    |   movel([-0.082267, -1.492529, -2.487581, -0.732279, 1.570796, 1.488530],accel_mss,speed_ms,0,blend_radius_m)
    |   movel([-0.082969, -1.494588, -2.485777, -0.732025, 1.570796, 1.487827],accel_mss,speed_ms,0,blend_radius_m)
    |   movel([-0.083539, -1.496624, -2.483986, -0.731779, 1.570796, 1.487258],accel_mss,speed_ms,0,blend_radius_m)
    |   movel([-0.083978, -1.498631, -2.482215, -0.731544, 1.570796, 1.486818],accel_mss,speed_ms,0,blend_radius_m)
    |   movel([-0.084285, -1.500606, -2.480465, -0.731318, 1.570796, 1.486511],accel_mss,speed_ms,0,blend_radius_m)
    |   movel([-0.084466, -1.502546, -2.478740, -0.731103, 1.570796, 1.486331],accel_mss,speed_ms,0,blend_radius_m)
    |   movel([-0.084516, -1.504447, -2.477045, -0.730898, 1.570796, 1.486280],accel_mss,speed_ms,0,blend_radius_m)
    |   movel([-0.084436, -1.506303, -2.475383, -0.730703, 1.570796, 1.486361],accel_mss,speed_ms,0,blend_radius_m)
    |   movel([-0.084230, -1.508115, -2.473757, -0.730518, 1.570796, 1.486566],accel_mss,speed_ms,0,blend_radius_m)
    |   movel([-0.083899, -1.509875, -2.472171, -0.730343, 1.570796, 1.486898],accel_mss,speed_ms,0,blend_radius_m)
    |   movel([-0.083438, -1.511581, -2.470630, -0.730178, 1.570796, 1.487358],accel_mss,speed_ms,0,blend_radius_m)
    |   movel([-0.082854, -1.513231, -2.469135, -0.730023, 1.570796, 1.487942],accel_mss,speed_ms,0,blend_radius_m)
    |   movel([-0.082145, -1.514819, -2.467691, -0.729879, 1.570796, 1.488651],accel_mss,speed_ms,0,blend_radius_m)
    |   movel([-0.081311, -1.516345, -2.466301, -0.729743, 1.570796, 1.489485],accel_mss,speed_ms,0,blend_radius_m)
    |   movel([-0.079795, -1.518566, -2.464270, -0.729553, 1.570796, 1.491001],accel_mss,speed_ms,0,blend_radius_m)
    |   movel([-0.078055, -1.520599, -2.462405, -0.729385, 1.570796, 1.492742],accel_mss,speed_ms,0,blend_radius_m)
    |   movel([-0.076117, -1.522459, -2.460692, -0.729238, 1.570796, 1.494679],accel_mss,speed_ms,0,blend_radius_m)
    |   movel([-0.074001, -1.524162, -2.459119, -0.729108, 1.570796, 1.496795],accel_mss,speed_ms,0,blend_radius_m)
    |   movel([-0.071735, -1.525724, -2.457672, -0.728993, 1.570796, 1.499062],accel_mss,speed_ms,0,blend_radius_m)
    |   movel([-0.069341, -1.527159, -2.456340, -0.728890, 1.570796, 1.501456],accel_mss,speed_ms,0,blend_radius_m)
    |   movel([-0.066843, -1.528483, -2.455108, -0.728799, 1.570796, 1.503953],accel_mss,speed_ms,0,blend_radius_m)
    |   movel([-0.064261, -1.529706, -2.453967, -0.728716, 1.570796, 1.506535],accel_mss,speed_ms,0,blend_radius_m)
    |   movel([-0.058915, -1.531954, -2.451863, -0.728572, 1.570796, 1.511882],accel_mss,speed_ms,0,blend_radius_m)
    |   movel([-0.053475, -1.534068, -2.449878, -0.728443, 1.570796, 1.517321],accel_mss,speed_ms,0,blend_radius_m)
    |   movel([-0.049350, -1.535795, -2.448251, -0.728343, 1.570796, 1.521446],accel_mss,speed_ms,0,blend_radius_m)
    |   movel([-0.047922, -1.536279, -2.447794, -0.728316, 1.570796, 1.522874],accel_mss,speed_ms,0,blend_radius_m)
    |   movel([-0.045334, -1.536940, -2.447169, -0.728280, 1.570796, 1.525463],accel_mss,speed_ms,0,blend_radius_m)
    |   movel([-0.044798, -1.537178, -2.446944, -0.728267, 1.570796, 1.525998],accel_mss,speed_ms,0,blend_radius_m)
    |   movel([-0.044322, -1.537503, -2.446637, -0.728250, 1.570796, 1.526475],accel_mss,speed_ms,0,blend_radius_m)
    |   movel([-0.043916, -1.537944, -2.446219, -0.728226, 1.570796, 1.526880],accel_mss,speed_ms,0,blend_radius_m)
    |   movel([-0.043592, -1.538530, -2.445663, -0.728195, 1.570796, 1.527205],accel_mss,speed_ms,0,blend_radius_m)
    |   movel([-0.043368, -1.539293, -2.444940, -0.728156, 1.570796, 1.527428],accel_mss,speed_ms,0,blend_radius_m)
    |   movel([-0.043314, -1.540103, -2.444171, -0.728116, 1.570796, 1.527483],accel_mss,speed_ms,0,blend_radius_m)
    |   movel([-0.043411, -1.540949, -2.443366, -0.728074, 1.570796, 1.527385],accel_mss,speed_ms,0,blend_radius_m)
    |   movel([-0.043649, -1.541827, -2.442530, -0.728033, 1.570796, 1.527148],accel_mss,speed_ms,0,blend_radius_m)
    |   movel([-0.044011, -1.542723, -2.441675, -0.727991, 1.570796, 1.526786],accel_mss,speed_ms,0,blend_radius_m)
    |   movel([-0.045056, -1.544546, -2.439931, -0.727912, 1.570796, 1.525740],accel_mss,speed_ms,0,blend_radius_m)
    |   movel([-0.045713, -1.545455, -2.439061, -0.727874, 1.570796, 1.525083],accel_mss,speed_ms,0,blend_radius_m)
    |   movel([-0.047218, -1.547224, -2.437361, -0.727804, 1.570796, 1.523578],accel_mss,speed_ms,0,blend_radius_m)
    |   movel([-0.048899, -1.548876, -2.435770, -0.727744, 1.570796, 1.521898],accel_mss,speed_ms,0,blend_radius_m)
    |   movel([-0.050641, -1.550343, -2.434352, -0.727694, 1.570796, 1.520155],accel_mss,speed_ms,0,blend_radius_m)
    |   movel([-0.052345, -1.551562, -2.433172, -0.727655, 1.570796, 1.518451],accel_mss,speed_ms,0,blend_radius_m)
    |   movel([-0.055003, -1.553125, -2.431656, -0.727608, 1.570796, 1.515794],accel_mss,speed_ms,0,blend_radius_m)
    |   movel([-0.056377, -1.553814, -2.430986, -0.727589, 1.570796, 1.514419],accel_mss,speed_ms,0,blend_radius_m)
    |   movel([-0.057771, -1.554438, -2.430379, -0.727572, 1.570796, 1.513025],accel_mss,speed_ms,0,blend_radius_m)
    |   movel([-0.060603, -1.555491, -2.429353, -0.727545, 1.570796, 1.510193],accel_mss,speed_ms,0,blend_radius_m)
    |   movel([-0.063453, -1.556276, -2.428587, -0.727526, 1.570796, 1.507344],accel_mss,speed_ms,0,blend_radius_m)
    |   movel([-0.066275, -1.556782, -2.428092, -0.727515, 1.570796, 1.504521],accel_mss,speed_ms,0,blend_radius_m)
    |   movel([-0.069020, -1.557000, -2.427879, -0.727510, 1.570796, 1.501776],accel_mss,speed_ms,0,blend_radius_m)
    |   movel([-0.070351, -1.556996, -2.427883, -0.727510, 1.570796, 1.500445],accel_mss,speed_ms,0,blend_radius_m)
    |   movel([-0.072900, -1.556759, -2.428115, -0.727515, 1.570796, 1.497896],accel_mss,speed_ms,0,blend_radius_m)
    |   movel([-0.074106, -1.556521, -2.428347, -0.727521, 1.570796, 1.496690],accel_mss,speed_ms,0,blend_radius_m)
    |   movel([-0.075629, -1.556091, -2.428768, -0.727531, 1.570796, 1.495168],accel_mss,speed_ms,0,blend_radius_m)
    |   movel([-0.077066, -1.555548, -2.429297, -0.727544, 1.570796, 1.493731],accel_mss,speed_ms,0,blend_radius_m)
    |   movel([-0.078425, -1.554908, -2.429921, -0.727560, 1.570796, 1.492372],accel_mss,speed_ms,0,blend_radius_m)
    |   movel([-0.079719, -1.554187, -2.430624, -0.727579, 1.570796, 1.491077],accel_mss,speed_ms,0,blend_radius_m)
    |   movel([-0.082152, -1.552560, -2.432204, -0.727624, 1.570796, 1.488644],accel_mss,speed_ms,0,blend_radius_m)
    |   movel([-0.084447, -1.550793, -2.433917, -0.727679, 1.570796, 1.486349],accel_mss,speed_ms,0,blend_radius_m)
    |   movel([-0.087214, -1.548474, -2.436157, -0.727758, 1.570796, 1.483583],accel_mss,speed_ms,0,blend_radius_m)
    |   movel([-0.089858, -1.546009, -2.438528, -0.727852, 1.570796, 1.480939],accel_mss,speed_ms,0,blend_radius_m)
    |   movel([-0.092354, -1.543396, -2.441032, -0.727961, 1.570796, 1.478443],accel_mss,speed_ms,0,blend_radius_m)
    |   movel([-0.094679, -1.540631, -2.443668, -0.728090, 1.570796, 1.476118],accel_mss,speed_ms,0,blend_radius_m)
    |   movel([-0.096807, -1.537710, -2.446441, -0.728238, 1.570796, 1.473989],accel_mss,speed_ms,0,blend_radius_m)
    |   movel([-0.098711, -1.534629, -2.449349, -0.728410, 1.570796, 1.472086],accel_mss,speed_ms,0,blend_radius_m)
    |   movel([-0.100365, -1.531386, -2.452395, -0.728608, 1.570796, 1.470431],accel_mss,speed_ms,0,blend_radius_m)
    |   movel([-0.101745, -1.527976, -2.455580, -0.728833, 1.570796, 1.469052],accel_mss,speed_ms,0,blend_radius_m)
    |   movel([-0.102598, -1.525304, -2.458061, -0.729023, 1.570796, 1.468199],accel_mss,speed_ms,0,blend_radius_m)
    |   movel([-0.103327, -1.522453, -2.460698, -0.729238, 1.570796, 1.467470],accel_mss,speed_ms,0,blend_radius_m)
    |   movel([-0.103895, -1.519449, -2.463461, -0.729479, 1.570796, 1.466901],accel_mss,speed_ms,0,blend_radius_m)
    |   movel([-0.104269, -1.516327, -2.466317, -0.729745, 1.570796, 1.466527],accel_mss,speed_ms,0,blend_radius_m)
    |   movel([-0.104412, -1.513119, -2.469236, -0.730034, 1.570796, 1.466384],accel_mss,speed_ms,0,blend_radius_m)
    |   movel([-0.104286, -1.509858, -2.472187, -0.730345, 1.570796, 1.466511],accel_mss,speed_ms,0,blend_radius_m)
    |   movel([-0.103856, -1.506574, -2.475141, -0.730675, 1.570796, 1.466940],accel_mss,speed_ms,0,blend_radius_m)
    |   movel([-0.103514, -1.504934, -2.476609, -0.730846, 1.570796, 1.467282],accel_mss,speed_ms,0,blend_radius_m)
    |   movel([-0.103083, -1.503302, -2.478066, -0.731020, 1.570796, 1.467714],accel_mss,speed_ms,0,blend_radius_m)
    |   movel([-0.102065, -1.500231, -2.480797, -0.731361, 1.570796, 1.468731],accel_mss,speed_ms,0,blend_radius_m)
    |   movel([-0.100816, -1.497139, -2.483531, -0.731718, 1.570796, 1.469980],accel_mss,speed_ms,0,blend_radius_m)
    |   movel([-0.099340, -1.494040, -2.486258, -0.732092, 1.570796, 1.471456],accel_mss,speed_ms,0,blend_radius_m)
    |   movel([-0.097645, -1.490946, -2.488963, -0.732480, 1.570796, 1.473151],accel_mss,speed_ms,0,blend_radius_m)
    |   movel([-0.095732, -1.487871, -2.491638, -0.732881, 1.570796, 1.475065],accel_mss,speed_ms,0,blend_radius_m)
    |   movel([-0.093611, -1.484830, -2.494267, -0.733292, 1.570796, 1.477185],accel_mss,speed_ms,0,blend_radius_m)
    |   movel([-0.091286, -1.481838, -2.496841, -0.733710, 1.570796, 1.479510],accel_mss,speed_ms,0,blend_radius_m)
    |   movel([-0.088762, -1.478910, -2.499346, -0.734134, 1.570796, 1.482034],accel_mss,speed_ms,0,blend_radius_m)
    |   movel([-0.092940, -1.473333, -2.504079, -0.734977, 1.570796, 1.477856],accel_mss,speed_ms,0,blend_radius_m)
    |   movel([-0.095041, -1.470536, -2.506435, -0.735418, 1.570796, 1.475755],accel_mss,speed_ms,0,blend_radius_m)
    |   movel([-0.097004, -1.467625, -2.508873, -0.735890, 1.570796, 1.473792],accel_mss,speed_ms,0,blend_radius_m)
    |   movel([-0.098264, -1.465308, -2.510805, -0.736276, 1.570796, 1.472533],accel_mss,speed_ms,0,blend_radius_m)
    |   movel([-0.099276, -1.462829, -2.512862, -0.736697, 1.570796, 1.471520],accel_mss,speed_ms,0,blend_radius_m)
    |   movel([-0.100052, -1.460205, -2.515030, -0.737154, 1.570796, 1.470745],accel_mss,speed_ms,0,blend_radius_m)
    |   movel([-0.100596, -1.457445, -2.517298, -0.737646, 1.570796, 1.470200],accel_mss,speed_ms,0,blend_radius_m)
    |   movel([-0.100917, -1.454564, -2.519654, -0.738172, 1.570796, 1.469879],accel_mss,speed_ms,0,blend_radius_m)
    |   movel([-0.101020, -1.451573, -2.522084, -0.738731, 1.570796, 1.469776],accel_mss,speed_ms,0,blend_radius_m)
    |   movel([-0.100913, -1.448486, -2.524579, -0.739323, 1.570796, 1.469883],accel_mss,speed_ms,0,blend_radius_m)
    |   movel([-0.100604, -1.445317, -2.527125, -0.739946, 1.570796, 1.470192],accel_mss,speed_ms,0,blend_radius_m)
    |   movel([-0.100098, -1.442082, -2.529709, -0.740598, 1.570796, 1.470699],accel_mss,speed_ms,0,blend_radius_m)
    |   movel([-0.099400, -1.438790, -2.532321, -0.741278, 1.570796, 1.471396],accel_mss,speed_ms,0,blend_radius_m)
    |   movel([-0.098520, -1.435458, -2.534948, -0.741983, 1.570796, 1.472277],accel_mss,speed_ms,0,blend_radius_m)
    |   movel([-0.097464, -1.432102, -2.537577, -0.742710, 1.570796, 1.473332],accel_mss,speed_ms,0,blend_radius_m)
    |   movel([-0.096240, -1.428735, -2.540197, -0.743456, 1.570796, 1.474556],accel_mss,speed_ms,0,blend_radius_m)
    |   movel([-0.094858, -1.425377, -2.542794, -0.744218, 1.570796, 1.475938],accel_mss,speed_ms,0,blend_radius_m)
    |   movel([-0.093321, -1.422040, -2.545357, -0.744992, 1.570796, 1.477475],accel_mss,speed_ms,0,blend_radius_m)
    |   movel([-0.091642, -1.418741, -2.547874, -0.745773, 1.570796, 1.479154],accel_mss,speed_ms,0,blend_radius_m)
    |   movel([-0.088194, -1.412581, -2.552532, -0.747276, 1.570796, 1.482602],accel_mss,speed_ms,0,blend_radius_m)
    |   movel([-0.086308, -1.409493, -2.554845, -0.748051, 1.570796, 1.484489],accel_mss,speed_ms,0,blend_radius_m)
    |   movel([-0.084288, -1.406418, -2.557135, -0.748837, 1.570796, 1.486508],accel_mss,speed_ms,0,blend_radius_m)
    |   movel([-0.082113, -1.403371, -2.559390, -0.749629, 1.570796, 1.488683],accel_mss,speed_ms,0,blend_radius_m)
    |   movel([-0.079766, -1.400370, -2.561597, -0.750422, 1.570796, 1.491030],accel_mss,speed_ms,0,blend_radius_m)
    |   movel([-0.077228, -1.397430, -2.563747, -0.751213, 1.570796, 1.493568],accel_mss,speed_ms,0,blend_radius_m)
    |   movel([-0.074479, -1.394567, -2.565828, -0.751994, 1.570796, 1.496318],accel_mss,speed_ms,0,blend_radius_m)
    |   movel([-0.071202, -1.391495, -2.568047, -0.752847, 1.570796, 1.499594],accel_mss,speed_ms,0,blend_radius_m)
    |   movel([-0.067735, -1.388536, -2.570172, -0.753681, 1.570796, 1.503061],accel_mss,speed_ms,0,blend_radius_m)
    |   movel([-0.064098, -1.385698, -2.572199, -0.754493, 1.570796, 1.506698],accel_mss,speed_ms,0,blend_radius_m)
    |   movel([-0.060310, -1.382989, -2.574122, -0.755278, 1.570796, 1.510487],accel_mss,speed_ms,0,blend_radius_m)
    |   movel([-0.056391, -1.380420, -2.575936, -0.756033, 1.570796, 1.514405],accel_mss,speed_ms,0,blend_radius_m)
    |   movel([-0.052365, -1.377999, -2.577636, -0.756753, 1.570796, 1.518431],accel_mss,speed_ms,0,blend_radius_m)
    |   movel([-0.048248, -1.375735, -2.579219, -0.757435, 1.570796, 1.522548],accel_mss,speed_ms,0,blend_radius_m)
    |   movel([-0.044065, -1.373638, -2.580679, -0.758072, 1.570796, 1.526731],accel_mss,speed_ms,0,blend_radius_m)
    |   movel([-0.039838, -1.371718, -2.582010, -0.758661, 1.570796, 1.530959],accel_mss,speed_ms,0,blend_radius_m)
    |   movel([-0.035590, -1.369980, -2.583210, -0.759199, 1.570796, 1.535206],accel_mss,speed_ms,0,blend_radius_m)
    |   movel([-0.031342, -1.368436, -2.584273, -0.759681, 1.570796, 1.539455],accel_mss,speed_ms,0,blend_radius_m)
    |   movel([-0.027115, -1.367091, -2.585195, -0.760103, 1.570796, 1.543681],accel_mss,speed_ms,0,blend_radius_m)
    |   movel([-0.022938, -1.365954, -2.585973, -0.760462, 1.570796, 1.547859],accel_mss,speed_ms,0,blend_radius_m)
    |   movel([-0.018827, -1.365032, -2.586603, -0.760754, 1.570796, 1.551969],accel_mss,speed_ms,0,blend_radius_m)
    |   movel([-0.014807, -1.364330, -2.587081, -0.760977, 1.570796, 1.555989],accel_mss,speed_ms,0,blend_radius_m)
    |   movel([-0.010899, -1.363858, -2.587403, -0.761128, 1.570796, 1.559897],accel_mss,speed_ms,0,blend_radius_m)
    |   movel([-0.006829, -1.363541, -2.587618, -0.761229, 1.570796, 1.563967],accel_mss,speed_ms,0,blend_radius_m)
    |   movel([-0.002820, -1.363384, -2.587726, -0.761280, 1.570796, 1.567976],accel_mss,speed_ms,0,blend_radius_m)
    |   movel([0.001098, -1.363425, -2.587697, -0.761266, 1.570796, 1.571894],accel_mss,speed_ms,0,blend_radius_m)
    |   movel([0.004894, -1.363713, -2.587502, -0.761175, 1.570796, 1.575691],accel_mss,speed_ms,0,blend_radius_m)
    |   movel([0.009149, -1.364394, -2.587038, -0.760957, 1.570796, 1.579946],accel_mss,speed_ms,0,blend_radius_m)
    |   movel([0.013233, -1.365436, -2.586327, -0.760626, 1.570796, 1.584029],accel_mss,speed_ms,0,blend_radius_m)
    |   movel([0.017106, -1.366821, -2.585380, -0.760188, 1.570796, 1.587902],accel_mss,speed_ms,0,blend_radius_m)
    |   movel([0.020731, -1.368531, -2.584207, -0.759651, 1.570796, 1.591527],accel_mss,speed_ms,0,blend_radius_m)
    |   movel([0.024074, -1.370546, -2.582819, -0.759024, 1.570796, 1.594870],accel_mss,speed_ms,0,blend_radius_m)
    |   movel([0.027099, -1.372846, -2.581228, -0.758315, 1.570796, 1.597895],accel_mss,speed_ms,0,blend_radius_m)
    |   movel([0.029775, -1.375406, -2.579449, -0.757534, 1.570796, 1.600572],accel_mss,speed_ms,0,blend_radius_m)
    |   movel([0.032074, -1.378207, -2.577491, -0.756691, 1.570796, 1.602870],accel_mss,speed_ms,0,blend_radius_m)
    |   movel([0.036161, -1.384036, -2.573380, -0.754973, 1.570796, 1.606957],accel_mss,speed_ms,0,blend_radius_m)
    |   movel([0.038008, -1.387050, -2.571235, -0.754104, 1.570796, 1.608804],accel_mss,speed_ms,0,blend_radius_m)
    |   movel([0.039646, -1.390258, -2.568937, -0.753194, 1.570796, 1.610442],accel_mss,speed_ms,0,blend_radius_m)
    |   movel([0.042293, -1.395720, -2.564991, -0.751678, 1.570796, 1.613089],accel_mss,speed_ms,0,blend_radius_m)
    |   movel([0.043799, -1.398370, -2.563061, -0.750959, 1.570796, 1.614595],accel_mss,speed_ms,0,blend_radius_m)
    |   movel([0.045476, -1.400889, -2.561216, -0.750284, 1.570796, 1.616272],accel_mss,speed_ms,0,blend_radius_m)
    |   movel([0.047368, -1.403223, -2.559499, -0.749667, 1.570796, 1.618164],accel_mss,speed_ms,0,blend_radius_m)
    |   movel([0.049508, -1.405317, -2.557951, -0.749121, 1.570796, 1.620304],accel_mss,speed_ms,0,blend_radius_m)
    |   movel([0.051940, -1.407117, -2.556616, -0.748657, 1.570796, 1.622736],accel_mss,speed_ms,0,blend_radius_m)
    |   movel([0.054700, -1.408569, -2.555535, -0.748286, 1.570796, 1.625496],accel_mss,speed_ms,0,blend_radius_m)
    |   movel([0.055929, -1.409007, -2.555208, -0.748174, 1.570796, 1.626726],accel_mss,speed_ms,0,blend_radius_m)
    |   movel([0.057287, -1.409249, -2.555027, -0.748113, 1.570796, 1.628084],accel_mss,speed_ms,0,blend_radius_m)
    |   movel([0.058007, -1.409257, -2.555021, -0.748111, 1.570796, 1.628803],accel_mss,speed_ms,0,blend_radius_m)
    |   movel([0.058747, -1.409170, -2.555086, -0.748133, 1.570796, 1.629544],accel_mss,speed_ms,0,blend_radius_m)
    |   movel([0.059507, -1.408974, -2.555233, -0.748183, 1.570796, 1.630304],accel_mss,speed_ms,0,blend_radius_m)
    |   movel([0.060279, -1.408650, -2.555474, -0.748265, 1.570796, 1.631075],accel_mss,speed_ms,0,blend_radius_m)
    |   movel([0.061049, -1.408194, -2.555814, -0.748381, 1.570796, 1.631845],accel_mss,speed_ms,0,blend_radius_m)
    |   movel([0.061762, -1.407642, -2.556225, -0.748522, 1.570796, 1.632558],accel_mss,speed_ms,0,blend_radius_m)
    |   movel([0.063014, -1.406358, -2.557179, -0.748852, 1.570796, 1.633811],accel_mss,speed_ms,0,blend_radius_m)
    |   movel([0.063753, -1.405394, -2.557894, -0.749101, 1.570796, 1.634550],accel_mss,speed_ms,0,blend_radius_m)
    |   movel([0.064381, -1.404409, -2.558623, -0.749357, 1.570796, 1.635177],accel_mss,speed_ms,0,blend_radius_m)
    |   movel([0.065330, -1.402399, -2.560106, -0.749884, 1.570796, 1.636126],accel_mss,speed_ms,0,blend_radius_m)
    |   movel([0.065915, -1.400362, -2.561603, -0.750424, 1.570796, 1.636712],accel_mss,speed_ms,0,blend_radius_m)
    |   movel([0.066194, -1.398329, -2.563090, -0.750970, 1.570796, 1.636991],accel_mss,speed_ms,0,blend_radius_m)
    |   movel([0.066220, -1.396340, -2.564540, -0.751509, 1.570796, 1.637016],accel_mss,speed_ms,0,blend_radius_m)
    |   movel([0.066047, -1.394428, -2.565928, -0.752033, 1.570796, 1.636844],accel_mss,speed_ms,0,blend_radius_m)
    |   movel([0.065732, -1.392629, -2.567230, -0.752531, 1.570796, 1.636528],accel_mss,speed_ms,0,blend_radius_m)
    |   movel([0.064746, -1.389183, -2.569709, -0.753497, 1.570796, 1.635542],accel_mss,speed_ms,0,blend_radius_m)
    |   movel([0.064002, -1.387475, -2.570931, -0.753983, 1.570796, 1.634799],accel_mss,speed_ms,0,blend_radius_m)
    |   movel([0.063104, -1.385861, -2.572082, -0.754446, 1.570796, 1.633900],accel_mss,speed_ms,0,blend_radius_m)
    |   movel([0.062052, -1.384355, -2.573153, -0.754881, 1.570796, 1.632848],accel_mss,speed_ms,0,blend_radius_m)
    |   movel([0.060847, -1.382961, -2.574142, -0.755287, 1.570796, 1.631643],accel_mss,speed_ms,0,blend_radius_m)
    |   movel([0.059493, -1.381691, -2.575039, -0.755658, 1.570796, 1.630289],accel_mss,speed_ms,0,blend_radius_m)
    |   movel([0.057997, -1.380552, -2.575842, -0.755994, 1.570796, 1.628794],accel_mss,speed_ms,0,blend_radius_m)
    |   movel([0.056359, -1.379553, -2.576545, -0.756290, 1.570796, 1.627155],accel_mss,speed_ms,0,blend_radius_m)
    |   speed_ms = 0.005
    |   movel([0.056359, -1.370765, -2.572549, -0.769076, 1.570796, 1.627155],accel_mss,speed_ms,0,blend_radius_m)
    |   speed_ms = 0.040
    |   movel([0.056256, -1.386026, -2.561797, -0.764566, 1.570796, 1.627052],accel_mss,speed_ms,0,blend_radius_m)
    |   speed_ms = 0.005
    |   movel([0.056256, -1.394705, -2.565727, -0.751956, 1.570796, 1.627052],accel_mss,speed_ms,0,blend_radius_m)
    |   speed_ms = 0.025
    |   movel([0.054176, -1.393655, -2.566488, -0.752246, 1.570796, 1.624973],accel_mss,speed_ms,0,blend_radius_m)
    |   movel([0.051871, -1.392874, -2.567053, -0.752462, 1.570796, 1.622668],accel_mss,speed_ms,0,blend_radius_m)
    |   movel([0.050615, -1.392653, -2.567212, -0.752524, 1.570796, 1.621411],accel_mss,speed_ms,0,blend_radius_m)
    |   movel([0.049282, -1.392584, -2.567262, -0.752543, 1.570796, 1.620078],accel_mss,speed_ms,0,blend_radius_m)
    |   movel([0.047868, -1.392691, -2.567184, -0.752513, 1.570796, 1.618664],accel_mss,speed_ms,0,blend_radius_m)
    |   movel([0.046364, -1.393002, -2.566960, -0.752427, 1.570796, 1.617160],accel_mss,speed_ms,0,blend_radius_m)
    |   speed_ms = 0.005
    |   movel([0.046364, -1.384310, -2.563022, -0.765057, 1.570796, 1.617160],accel_mss,speed_ms,0,blend_radius_m)
    |   speed_ms = 0.040
    |   movel([0.050800, -1.379714, -2.566284, -0.766391, 1.570796, 1.621596],accel_mss,speed_ms,0,blend_radius_m)
    |   speed_ms = 0.005
    |   movel([0.050800, -1.388439, -2.570242, -0.753708, 1.570796, 1.621596],accel_mss,speed_ms,0,blend_radius_m)
    |   speed_ms = 0.025
    |   movel([0.050701, -1.386443, -2.571668, -0.754278, 1.570796, 1.621498],accel_mss,speed_ms,0,blend_radius_m)
    |   movel([0.050175, -1.384681, -2.572921, -0.754786, 1.570796, 1.620971],accel_mss,speed_ms,0,blend_radius_m)
    |   movel([0.049255, -1.383178, -2.573988, -0.755223, 1.570796, 1.620052],accel_mss,speed_ms,0,blend_radius_m)
    |   movel([0.047974, -1.381967, -2.574845, -0.755578, 1.570796, 1.618770],accel_mss,speed_ms,0,blend_radius_m)
    |   movel([0.046366, -1.381074, -2.575475, -0.755840, 1.570796, 1.617163],accel_mss,speed_ms,0,blend_radius_m)
    |   movel([0.044470, -1.380530, -2.575858, -0.756001, 1.570796, 1.615267],accel_mss,speed_ms,0,blend_radius_m)
    |   movel([0.042323, -1.380360, -2.575978, -0.756051, 1.570796, 1.613120],accel_mss,speed_ms,0,blend_radius_m)
    |   movel([0.041166, -1.380425, -2.575932, -0.756032, 1.570796, 1.611962],accel_mss,speed_ms,0,blend_radius_m)
    |   movel([0.039961, -1.380591, -2.575815, -0.755983, 1.570796, 1.610757],accel_mss,speed_ms,0,blend_radius_m)
    |   speed_ms = 0.005
    |   movel([0.039961, -1.371810, -2.571823, -0.768756, 1.570796, 1.610757],accel_mss,speed_ms,0,blend_radius_m)
    |   speed_ms = 0.040
    |   movel([0.045655, -1.367633, -2.574714, -0.770042, 1.570796, 1.616452],accel_mss,speed_ms,0,blend_radius_m)
    |   speed_ms = 0.005
    |   movel([0.045655, -1.376444, -2.578724, -0.757221, 1.570796, 1.616452],accel_mss,speed_ms,0,blend_radius_m)
    |   speed_ms = 0.025
    |   movel([0.045426, -1.375518, -2.579371, -0.757501, 1.570796, 1.616223],accel_mss,speed_ms,0,blend_radius_m)
    |   movel([0.045059, -1.374646, -2.579978, -0.757765, 1.570796, 1.615855],accel_mss,speed_ms,0,blend_radius_m)
    |   movel([0.043947, -1.373084, -2.581063, -0.758242, 1.570796, 1.614743],accel_mss,speed_ms,0,blend_radius_m)
    |   movel([0.042397, -1.371794, -2.581957, -0.758638, 1.570796, 1.613193],accel_mss,speed_ms,0,blend_radius_m)
    |   movel([0.040492, -1.370817, -2.582633, -0.758940, 1.570796, 1.611289],accel_mss,speed_ms,0,blend_radius_m)
    |   movel([0.038312, -1.370180, -2.583072, -0.759137, 1.570796, 1.609108],accel_mss,speed_ms,0,blend_radius_m)
    |   movel([0.035947, -1.369917, -2.583253, -0.759219, 1.570796, 1.606743],accel_mss,speed_ms,0,blend_radius_m)
    |   movel([0.034719, -1.369938, -2.583239, -0.759212, 1.570796, 1.605515],accel_mss,speed_ms,0,blend_radius_m)
    |   movel([0.032231, -1.370296, -2.582992, -0.759101, 1.570796, 1.603027],accel_mss,speed_ms,0,blend_radius_m)
    |   movel([0.030992, -1.370640, -2.582755, -0.758995, 1.570796, 1.601788],accel_mss,speed_ms,0,blend_radius_m)
    |   speed_ms = 0.005
    |   movel([0.030992, -1.361788, -2.578719, -0.771882, 1.570796, 1.601788],accel_mss,speed_ms,0,blend_radius_m)
    |   speed_ms = 0.040
    |   movel([0.039126, -1.356851, -2.582064, -0.773474, 1.570796, 1.609923],accel_mss,speed_ms,0,blend_radius_m)
    |   speed_ms = 0.005
    |   movel([0.039126, -1.365737, -2.586122, -0.760531, 1.570796, 1.609923],accel_mss,speed_ms,0,blend_radius_m)
    |   speed_ms = 0.025
    |   movel([0.037538, -1.364150, -2.587204, -0.761035, 1.570796, 1.608334],accel_mss,speed_ms,0,blend_radius_m)
    |   movel([0.035621, -1.362863, -2.588079, -0.761446, 1.570796, 1.606418],accel_mss,speed_ms,0,blend_radius_m)
    |   movel([0.033416, -1.361920, -2.588719, -0.761750, 1.570796, 1.604213],accel_mss,speed_ms,0,blend_radius_m)
    |   movel([0.030951, -1.361352, -2.589104, -0.761933, 1.570796, 1.601747],accel_mss,speed_ms,0,blend_radius_m)
    |   movel([0.028264, -1.361199, -2.589207, -0.761982, 1.570796, 1.599060],accel_mss,speed_ms,0,blend_radius_m)
    |   movel([0.026848, -1.361288, -2.589147, -0.761954, 1.570796, 1.597645],accel_mss,speed_ms,0,blend_radius_m)
    |   movel([0.025393, -1.361494, -2.589008, -0.761887, 1.570796, 1.596189],accel_mss,speed_ms,0,blend_radius_m)
    |   movel([0.023898, -1.361820, -2.588787, -0.761782, 1.570796, 1.594695],accel_mss,speed_ms,0,blend_radius_m)
    |   movel([0.022370, -1.362271, -2.588481, -0.761637, 1.570796, 1.593166],accel_mss,speed_ms,0,blend_radius_m)
    |   movel([0.020816, -1.362849, -2.588089, -0.761451, 1.570796, 1.591612],accel_mss,speed_ms,0,blend_radius_m)
    |   movel([0.019239, -1.363559, -2.587606, -0.761224, 1.570796, 1.590036],accel_mss,speed_ms,0,blend_radius_m)
    |   speed_ms = 0.005
    |   movel([0.019239, -1.354658, -2.583539, -0.774192, 1.570796, 1.590036],accel_mss,speed_ms,0,blend_radius_m)
    |   speed_ms = 0.040
    |   movel([0.027863, -1.348222, -2.587830, -0.776338, 1.570796, 1.598660],accel_mss,speed_ms,0,blend_radius_m)
    |   speed_ms = 0.005
    |   movel([0.027863, -1.357166, -2.591926, -0.763297, 1.570796, 1.598660],accel_mss,speed_ms,0,blend_radius_m)
    |   speed_ms = 0.025
    |   movel([0.027318, -1.355873, -2.592792, -0.763723, 1.570796, 1.598114],accel_mss,speed_ms,0,blend_radius_m)
    |   movel([0.026528, -1.354745, -2.593546, -0.764097, 1.570796, 1.597324],accel_mss,speed_ms,0,blend_radius_m)
    |   movel([0.025508, -1.353804, -2.594174, -0.764410, 1.570796, 1.596304],accel_mss,speed_ms,0,blend_radius_m)
    |   movel([0.024278, -1.353073, -2.594661, -0.764655, 1.570796, 1.595074],accel_mss,speed_ms,0,blend_radius_m)
    |   movel([0.022555, -1.352476, -2.595058, -0.764855, 1.570796, 1.593351],accel_mss,speed_ms,0,blend_radius_m)
    |   movel([0.020651, -1.352134, -2.595285, -0.764969, 1.570796, 1.591447],accel_mss,speed_ms,0,blend_radius_m)
    |   movel([0.018265, -1.351979, -2.595389, -0.765022, 1.570796, 1.589062],accel_mss,speed_ms,0,blend_radius_m)
    |   movel([0.015752, -1.352104, -2.595306, -0.764980, 1.570796, 1.586548],accel_mss,speed_ms,0,blend_radius_m)
    |   movel([0.013143, -1.352538, -2.595017, -0.764834, 1.570796, 1.583939],accel_mss,speed_ms,0,blend_radius_m)
    |   movel([0.010469, -1.353317, -2.594499, -0.764573, 1.570796, 1.581266],accel_mss,speed_ms,0,blend_radius_m)
    |   movel([0.007776, -1.354471, -2.593729, -0.764188, 1.570796, 1.578573],accel_mss,speed_ms,0,blend_radius_m)
    |   movel([0.006451, -1.355185, -2.593253, -0.763951, 1.570796, 1.577247],accel_mss,speed_ms,0,blend_radius_m)
    |   movel([0.003913, -1.356864, -2.592129, -0.763397, 1.570796, 1.574709],accel_mss,speed_ms,0,blend_radius_m)
    |   movel([0.002724, -1.357817, -2.591488, -0.763083, 1.570796, 1.573520],accel_mss,speed_ms,0,blend_radius_m)
    |   movel([0.001609, -1.358842, -2.590799, -0.762748, 1.570796, 1.572406],accel_mss,speed_ms,0,blend_radius_m)
    |   movel([0.000580, -1.359933, -2.590063, -0.762392, 1.570796, 1.571376],accel_mss,speed_ms,0,blend_radius_m)
    |   speed_ms = 0.005
    |   movel([0.000580, -1.351007, -2.585980, -0.775402, 1.570796, 1.571376],accel_mss,speed_ms,0,blend_radius_m)
    |   speed_ms = 0.040
    |   movel([0.009787, -1.340894, -2.592645, -0.778850, 1.570796, 1.580584],accel_mss,speed_ms,0,blend_radius_m)
    |   speed_ms = 0.005
    |   movel([0.009787, -1.349888, -2.596774, -0.765727, 1.570796, 1.580584],accel_mss,speed_ms,0,blend_radius_m)
    |   speed_ms = 0.025
    |   movel([0.006644, -1.349839, -2.596806, -0.765744, 1.570796, 1.577440],accel_mss,speed_ms,0,blend_radius_m)
    |   movel([0.003301, -1.350135, -2.596610, -0.765644, 1.570796, 1.574097],accel_mss,speed_ms,0,blend_radius_m)
    |   movel([-0.000160, -1.350811, -2.596163, -0.765415, 1.570796, 1.570637],accel_mss,speed_ms,0,blend_radius_m)
    |   movel([-0.001908, -1.351297, -2.595841, -0.765251, 1.570796, 1.568888],accel_mss,speed_ms,0,blend_radius_m)
    |   movel([-0.003655, -1.351890, -2.595448, -0.765052, 1.570796, 1.567141],accel_mss,speed_ms,0,blend_radius_m)
    |   movel([-0.005388, -1.352589, -2.594983, -0.764817, 1.570796, 1.565409],accel_mss,speed_ms,0,blend_radius_m)
    |   movel([-0.007094, -1.353398, -2.594445, -0.764546, 1.570796, 1.563702],accel_mss,speed_ms,0,blend_radius_m)
    |   movel([-0.008766, -1.354321, -2.593829, -0.764238, 1.570796, 1.562031],accel_mss,speed_ms,0,blend_radius_m)
    |   movel([-0.010392, -1.355362, -2.593134, -0.763893, 1.570796, 1.560405],accel_mss,speed_ms,0,blend_radius_m)
    |   movel([-0.011963, -1.356521, -2.592359, -0.763510, 1.570796, 1.558833],accel_mss,speed_ms,0,blend_radius_m)
    |   movel([-0.013464, -1.357801, -2.591499, -0.763088, 1.570796, 1.557332],accel_mss,speed_ms,0,blend_radius_m)
    |   movel([-0.014889, -1.359205, -2.590555, -0.762630, 1.570796, 1.555907],accel_mss,speed_ms,0,blend_radius_m)
    |   movel([-0.016224, -1.360736, -2.589521, -0.762132, 1.570796, 1.554572],accel_mss,speed_ms,0,blend_radius_m)
    |   speed_ms = 0.005
    |   movel([-0.016224, -1.351815, -2.585441, -0.775133, 1.570796, 1.554572],accel_mss,speed_ms,0,blend_radius_m)
    |   speed_ms = 0.040
    |   movel([-0.009624, -1.340342, -2.593005, -0.779042, 1.570796, 1.561172],accel_mss,speed_ms,0,blend_radius_m)
    |   speed_ms = 0.005
    |   movel([-0.009624, -1.349340, -2.597136, -0.765913, 1.570796, 1.561172],accel_mss,speed_ms,0,blend_radius_m)
    |   speed_ms = 0.025
    |   movel([-0.011251, -1.349433, -2.597074, -0.765882, 1.570796, 1.559545],accel_mss,speed_ms,0,blend_radius_m)
    |   movel([-0.012933, -1.349679, -2.596912, -0.765798, 1.570796, 1.557864],accel_mss,speed_ms,0,blend_radius_m)
    |   movel([-0.014648, -1.350076, -2.596650, -0.765664, 1.570796, 1.556148],accel_mss,speed_ms,0,blend_radius_m)
    |   movel([-0.016385, -1.350614, -2.596294, -0.765482, 1.570796, 1.554412],accel_mss,speed_ms,0,blend_radius_m)
    |   movel([-0.018128, -1.351290, -2.595846, -0.765254, 1.570796, 1.552669],accel_mss,speed_ms,0,blend_radius_m)
    |   movel([-0.019858, -1.352097, -2.595310, -0.764982, 1.570796, 1.550938],accel_mss,speed_ms,0,blend_radius_m)
    |   movel([-0.021560, -1.353028, -2.594691, -0.764670, 1.570796, 1.549236],accel_mss,speed_ms,0,blend_radius_m)
    |   movel([-0.023221, -1.354078, -2.593992, -0.764319, 1.570796, 1.547575],accel_mss,speed_ms,0,blend_radius_m)
    |   movel([-0.024821, -1.355239, -2.593217, -0.763933, 1.570796, 1.545975],accel_mss,speed_ms,0,blend_radius_m)
    |   movel([-0.026346, -1.356495, -2.592376, -0.763518, 1.570796, 1.544450],accel_mss,speed_ms,0,blend_radius_m)
    |   movel([-0.027783, -1.357833, -2.591478, -0.763078, 1.570796, 1.543013],accel_mss,speed_ms,0,blend_radius_m)
    |   movel([-0.029122, -1.359241, -2.590530, -0.762618, 1.570796, 1.541674],accel_mss,speed_ms,0,blend_radius_m)
    |   movel([-0.030353, -1.360704, -2.589543, -0.762143, 1.570796, 1.540443],accel_mss,speed_ms,0,blend_radius_m)
    |   movel([-0.031466, -1.362211, -2.588522, -0.761656, 1.570796, 1.539331],accel_mss,speed_ms,0,blend_radius_m)
    |   movel([-0.032443, -1.363746, -2.587479, -0.761164, 1.570796, 1.538354],accel_mss,speed_ms,0,blend_radius_m)
    |   movel([-0.033280, -1.365298, -2.586422, -0.760670, 1.570796, 1.537516],accel_mss,speed_ms,0,blend_radius_m)
    |   speed_ms = 0.005
    |   movel([-0.033280, -1.356409, -2.582362, -0.773618, 1.570796, 1.537516],accel_mss,speed_ms,0,blend_radius_m)
    |   speed_ms = 0.040
    |   movel([-0.029508, -1.345457, -2.589655, -0.777277, 1.570796, 1.541288],accel_mss,speed_ms,0,blend_radius_m)
    |   speed_ms = 0.005
    |   movel([-0.029508, -1.354421, -2.593763, -0.764205, 1.570796, 1.541288],accel_mss,speed_ms,0,blend_radius_m)
    |   speed_ms = 0.025
    |   movel([-0.031119, -1.354616, -2.593633, -0.764140, 1.570796, 1.539678],accel_mss,speed_ms,0,blend_radius_m)
    |   movel([-0.032775, -1.355067, -2.593332, -0.763991, 1.570796, 1.538021],accel_mss,speed_ms,0,blend_radius_m)
    |   movel([-0.034448, -1.355742, -2.592880, -0.763767, 1.570796, 1.536348],accel_mss,speed_ms,0,blend_radius_m)
    |   movel([-0.036120, -1.356609, -2.592299, -0.763480, 1.570796, 1.534677],accel_mss,speed_ms,0,blend_radius_m)
    |   movel([-0.037765, -1.357638, -2.591609, -0.763142, 1.570796, 1.533031],accel_mss,speed_ms,0,blend_radius_m)
    |   movel([-0.039359, -1.358795, -2.590831, -0.762763, 1.570796, 1.531437],accel_mss,speed_ms,0,blend_radius_m)
    |   movel([-0.040885, -1.360047, -2.589986, -0.762356, 1.570796, 1.529911],accel_mss,speed_ms,0,blend_radius_m)
    |   movel([-0.042314, -1.361365, -2.589095, -0.761929, 1.570796, 1.528483],accel_mss,speed_ms,0,blend_radius_m)
    |   movel([-0.043694, -1.362780, -2.588136, -0.761473, 1.570796, 1.527102],accel_mss,speed_ms,0,blend_radius_m)
    |   movel([-0.044980, -1.364256, -2.587132, -0.761001, 1.570796, 1.525816],accel_mss,speed_ms,0,blend_radius_m)
    |   movel([-0.046152, -1.365777, -2.586094, -0.760518, 1.570796, 1.524645],accel_mss,speed_ms,0,blend_radius_m)
    |   movel([-0.047176, -1.367326, -2.585034, -0.760029, 1.570796, 1.523620],accel_mss,speed_ms,0,blend_radius_m)
    |   movel([-0.048032, -1.368882, -2.583966, -0.759541, 1.570796, 1.522765],accel_mss,speed_ms,0,blend_radius_m)
    |   movel([-0.048694, -1.370427, -2.582901, -0.759060, 1.570796, 1.522103],accel_mss,speed_ms,0,blend_radius_m)
    |   movel([-0.049130, -1.371946, -2.581852, -0.758591, 1.570796, 1.521666],accel_mss,speed_ms,0,blend_radius_m)
    |   movel([-0.049322, -1.373418, -2.580832, -0.758139, 1.570796, 1.521474],accel_mss,speed_ms,0,blend_radius_m)
    |   speed_ms = 0.005
    |   movel([-0.049322, -1.364586, -2.576808, -0.770995, 1.570796, 1.521474],accel_mss,speed_ms,0,blend_radius_m)
    |   speed_ms = 0.040
    |   movel([-0.049808, -1.355807, -2.582767, -0.773815, 1.570796, 1.520988],accel_mss,speed_ms,0,blend_radius_m)
    |   speed_ms = 0.005
    |   movel([-0.049808, -1.364700, -2.586829, -0.760859, 1.570796, 1.520988],accel_mss,speed_ms,0,blend_radius_m)
    |   speed_ms = 0.025
    |   movel([-0.052106, -1.366060, -2.585901, -0.760428, 1.570796, 1.518691],accel_mss,speed_ms,0,blend_radius_m)
    |   movel([-0.054439, -1.367711, -2.584770, -0.759908, 1.570796, 1.516358],accel_mss,speed_ms,0,blend_radius_m)
    |   movel([-0.056681, -1.369587, -2.583480, -0.759321, 1.570796, 1.514116],accel_mss,speed_ms,0,blend_radius_m)
    |   movel([-0.058703, -1.371619, -2.582078, -0.758692, 1.570796, 1.512093],accel_mss,speed_ms,0,blend_radius_m)
    |   movel([-0.060386, -1.373741, -2.580607, -0.758041, 1.570796, 1.510411],accel_mss,speed_ms,0,blend_radius_m)
    |   movel([-0.061062, -1.374817, -2.579859, -0.757713, 1.570796, 1.509735],accel_mss,speed_ms,0,blend_radius_m)
    |   movel([-0.061605, -1.375890, -2.579111, -0.757388, 1.570796, 1.509191],accel_mss,speed_ms,0,blend_radius_m)
    |   movel([-0.062005, -1.376955, -2.578367, -0.757067, 1.570796, 1.508792],accel_mss,speed_ms,0,blend_radius_m)
    |   movel([-0.062245, -1.378004, -2.577633, -0.756752, 1.570796, 1.508551],accel_mss,speed_ms,0,blend_radius_m)
    |   movel([-0.062307, -1.379024, -2.576917, -0.756447, 1.570796, 1.508490],accel_mss,speed_ms,0,blend_radius_m)
    |   movel([-0.062180, -1.380016, -2.576220, -0.756153, 1.570796, 1.508616],accel_mss,speed_ms,0,blend_radius_m)
    |   speed_ms = 0.005
    |   movel([-0.062180, -1.371230, -2.572225, -0.768933, 1.570796, 1.508616],accel_mss,speed_ms,0,blend_radius_m)
    |   speed_ms = 0.040
    |   movel([-0.066185, -1.368693, -2.573983, -0.769713, 1.570796, 1.504611],accel_mss,speed_ms,0,blend_radius_m)
    |   speed_ms = 0.005
    |   movel([-0.066185, -1.377496, -2.577989, -0.756904, 1.570796, 1.504611],accel_mss,speed_ms,0,blend_radius_m)
    |   speed_ms = 0.025
    |   movel([-0.068894, -1.380459, -2.575908, -0.756022, 1.570796, 1.501902],accel_mss,speed_ms,0,blend_radius_m)
    |   movel([-0.070132, -1.382012, -2.574813, -0.755564, 1.570796, 1.500664],accel_mss,speed_ms,0,blend_radius_m)
    |   movel([-0.071233, -1.383588, -2.573697, -0.755104, 1.570796, 1.499563],accel_mss,speed_ms,0,blend_radius_m)
    |   movel([-0.072155, -1.385178, -2.572568, -0.754642, 1.570796, 1.498642],accel_mss,speed_ms,0,blend_radius_m)
    |   movel([-0.072857, -1.386769, -2.571435, -0.754185, 1.570796, 1.497939],accel_mss,speed_ms,0,blend_radius_m)
    |   movel([-0.073294, -1.388344, -2.570309, -0.753735, 1.570796, 1.497502],accel_mss,speed_ms,0,blend_radius_m)
    |   movel([-0.073429, -1.389895, -2.569198, -0.753296, 1.570796, 1.497368],accel_mss,speed_ms,0,blend_radius_m)
    |   speed_ms = 0.005
    |   # Splitting Linear movement in 2 (instruction 3386: MoveL 3110)
    |   movel([-0.073429, -1.368405, -2.559208, -0.784776, 1.570796, 1.497368],accel_mss,speed_ms,0,blend_radius_m)
    |   movel([-0.073429, -1.347892, -2.548856, -0.815641, 1.570796, 1.497368],accel_mss,speed_ms,0,blend_radius_m)
    |   speed_ms = 1.000
    |   movel([-0.073429, -1.347892, -2.548856, -0.815641, 1.570796, 1.497368],accel_mss,speed_ms,0,blend_radius_m)
    |   # Splitting Linear movement in 2 (instruction 3389: MoveL 3112)
    |   movel([-0.073429, -1.318924, -2.532681, -0.860784, 1.570796, 1.497368],accel_mss,speed_ms,0,blend_radius_m)
    |   movel([-0.073429, -1.292060, -2.515776, -0.904553, 1.570796, 1.497368],accel_mss,speed_ms,0,blend_radius_m)
    |   # End of main program
    | end
    | 
    | Machining2()
  Script file /programs/usbdisk_0/azat/test_fourth_drawing_8_m18.script
    | def Machining4():
    |   # Default parameters:
    |   global speed_ms = 0.3
    |   global speed_rads = 0.75
    |   global accel_mss = 3
    |   global accel_radss = 1.2
    |   global blend_radius_m = 0.001
    | 
    |   # Add subprograms here
    |   # Start of main program
    |   # Program generated by RoboDK v5.6.5 for UR10e on 02/02/2024 17:39:49
    |   # Using nominal kinematics.
    |   blend_radius_m = 0.001
    |   speed_ms = 1.000
    |   # set_reference(p[0.348734, -0.005000, -0.017586, 0.000000, 0.000000, 0.000000])
    |   set_tcp(p[0.000000, 0.000000, 0.252000, 0.000000, 0.000000, 0.000000])
    |   # Show Tool
    |   movej([0.508484, -0.952512, -2.535391, -1.224486, 1.570796, 2.079280],accel_radss,speed_rads,0,blend_radius_m)
    |   movel([0.508484, -0.952512, -2.535391, -1.224486, 1.570796, 2.079280],accel_mss,speed_ms,0,blend_radius_m)
    |   # Splitting Linear movement in 6 (instruction 7: MoveL 3)
    |   movel([0.508484, -0.969998, -2.560672, -1.181720, 1.570796, 2.079280],accel_mss,speed_ms,0,blend_radius_m)
    |   movel([0.508484, -0.990214, -2.585461, -1.136714, 1.570796, 2.079280],accel_mss,speed_ms,0,blend_radius_m)
    |   movel([0.508484, -1.013449, -2.609714, -1.089227, 1.570796, 2.079280],accel_mss,speed_ms,0,blend_radius_m)
    |   movel([0.508484, -1.040019, -2.633377, -1.038993, 1.570796, 2.079280],accel_mss,speed_ms,0,blend_radius_m)
    |   movel([0.508484, -1.070270, -2.656387, -0.985731, 1.570796, 2.079280],accel_mss,speed_ms,0,blend_radius_m)
    |   movel([0.508484, -1.104577, -2.678669, -0.929143, 1.570796, 2.079280],accel_mss,speed_ms,0,blend_radius_m)
    |   movel([0.508484, -1.104577, -2.678669, -0.929143, 1.570796, 2.079280],accel_mss,speed_ms,0,blend_radius_m)
    |   speed_ms = 1.000
    |   movel([0.508484, -1.104577, -2.678669, -0.929143, 1.570796, 2.079280],accel_mss,speed_ms,0,blend_radius_m)
    |   movel([0.508484, -1.104577, -2.678669, -0.929143, 1.570796, 2.079280],accel_mss,speed_ms,0,blend_radius_m)
    |   movel([0.508484, -1.104577, -2.678669, -0.929143, 1.570796, 2.079280],accel_mss,speed_ms,0,blend_radius_m)
    |   speed_ms = 0.005
    |   movel([0.508484, -1.063908, -2.651841, -0.996640, 1.570796, 2.079280],accel_mss,speed_ms,0,blend_radius_m)
    |   speed_ms = 1.000
    |   movel([0.508484, -1.104577, -2.678669, -0.929143, 1.570796, 2.079280],accel_mss,speed_ms,0,blend_radius_m)
    |   speed_ms = 0.040
    |   movel([0.508484, -1.104577, -2.678669, -0.929143, 1.570796, 2.079280],accel_mss,speed_ms,0,blend_radius_m)
    |   speed_ms = 1.000
    |   movel([0.508484, -1.104577, -2.678669, -0.929143, 1.570796, 2.079280],accel_mss,speed_ms,0,blend_radius_m)
    |   # Splitting Linear movement in 8 (instruction 21: MoveL 12)
    |   movel([0.516357, -1.145060, -2.661765, -0.905563, 1.570796, 2.087153],accel_mss,speed_ms,0,blend_radius_m)
    |   movel([0.523521, -1.183921, -2.644010, -0.884457, 1.570796, 2.094317],accel_mss,speed_ms,0,blend_radius_m)
    |   movel([0.530064, -1.221217, -2.625467, -0.865705, 1.570796, 2.100861],accel_mss,speed_ms,0,blend_radius_m)
    |   movel([0.536061, -1.257021, -2.606194, -0.849174, 1.570796, 2.106857],accel_mss,speed_ms,0,blend_radius_m)
    |   movel([0.541574, -1.291418, -2.586246, -0.834725, 1.570796, 2.112371],accel_mss,speed_ms,0,blend_radius_m)
    |   movel([0.546659, -1.324498, -2.565672, -0.822220, 1.570796, 2.117455],accel_mss,speed_ms,0,blend_radius_m)
    |   movel([0.551360, -1.356351, -2.544515, -0.811522, 1.570796, 2.122157],accel_mss,speed_ms,0,blend_radius_m)
    |   movel([0.555720, -1.387070, -2.522816, -0.802503, 1.570796, 2.126517],accel_mss,speed_ms,0,blend_radius_m)
    |   speed_ms = 0.005
    |   movel([0.555720, -1.427952, -2.542321, -0.742116, 1.570796, 2.126517],accel_mss,speed_ms,0,blend_radius_m)
    |   speed_ms = 0.025
    |   movel([0.551886, -1.431799, -2.539331, -0.741259, 1.570796, 2.122682],accel_mss,speed_ms,0,blend_radius_m)
    |   movel([0.549891, -1.433665, -2.537873, -0.740851, 1.570796, 2.120688],accel_mss,speed_ms,0,blend_radius_m)
    |   movel([0.547837, -1.435468, -2.536459, -0.740462, 1.570796, 2.118634],accel_mss,speed_ms,0,blend_radius_m)
    |   movel([0.545720, -1.437189, -2.535105, -0.740095, 1.570796, 2.116517],accel_mss,speed_ms,0,blend_radius_m)
    |   movel([0.543536, -1.438810, -2.533826, -0.739753, 1.570796, 2.114332],accel_mss,speed_ms,0,blend_radius_m)
    |   movel([0.541277, -1.440313, -2.532636, -0.739441, 1.570796, 2.112073],accel_mss,speed_ms,0,blend_radius_m)
    |   movel([0.538938, -1.441676, -2.531553, -0.739160, 1.570796, 2.109734],accel_mss,speed_ms,0,blend_radius_m)
    |   movel([0.539897, -1.440992, -2.532097, -0.739300, 1.570796, 2.110693],accel_mss,speed_ms,0,blend_radius_m)
    |   movel([0.540974, -1.439974, -2.532904, -0.739511, 1.570796, 2.111771],accel_mss,speed_ms,0,blend_radius_m)
    |   movel([0.541871, -1.438872, -2.533777, -0.739741, 1.570796, 2.112668],accel_mss,speed_ms,0,blend_radius_m)
    |   movel([0.542155, -1.438369, -2.534174, -0.739846, 1.570796, 2.112951],accel_mss,speed_ms,0,blend_radius_m)
    |   movel([0.542280, -1.437941, -2.534512, -0.739936, 1.570796, 2.113076],accel_mss,speed_ms,0,blend_radius_m)
    |   movel([0.542211, -1.437608, -2.534775, -0.740006, 1.570796, 2.113008],accel_mss,speed_ms,0,blend_radius_m)
    |   movel([0.541951, -1.437454, -2.534896, -0.740039, 1.570796, 2.112747],accel_mss,speed_ms,0,blend_radius_m)
    |   movel([0.541528, -1.437461, -2.534891, -0.740037, 1.570796, 2.112324],accel_mss,speed_ms,0,blend_radius_m)
    |   movel([0.540960, -1.437607, -2.534776, -0.740007, 1.570796, 2.111756],accel_mss,speed_ms,0,blend_radius_m)
    |   movel([0.539505, -1.438234, -2.534280, -0.739874, 1.570796, 2.110301],accel_mss,speed_ms,0,blend_radius_m)
    |   movel([0.537786, -1.439172, -2.533539, -0.739678, 1.570796, 2.108582],accel_mss,speed_ms,0,blend_radius_m)
    |   movel([0.534336, -1.441332, -2.531826, -0.739230, 1.570796, 2.105133],accel_mss,speed_ms,0,blend_radius_m)
    |   movel([0.532176, -1.442774, -2.530679, -0.738936, 1.570796, 2.102972],accel_mss,speed_ms,0,blend_radius_m)
    |   movel([0.529059, -1.444697, -2.529144, -0.738548, 1.570796, 2.099855],accel_mss,speed_ms,0,blend_radius_m)
    |   movel([0.527463, -1.445498, -2.528503, -0.738388, 1.570796, 2.098260],accel_mss,speed_ms,0,blend_radius_m)
    |   movel([0.525843, -1.446095, -2.528025, -0.738269, 1.570796, 2.096640],accel_mss,speed_ms,0,blend_radius_m)
    |   movel([0.526257, -1.445821, -2.528245, -0.738324, 1.570796, 2.097053],accel_mss,speed_ms,0,blend_radius_m)
    |   movel([0.526732, -1.445268, -2.528687, -0.738434, 1.570796, 2.097529],accel_mss,speed_ms,0,blend_radius_m)
    |   movel([0.527721, -1.443665, -2.529968, -0.738755, 1.570796, 2.098517],accel_mss,speed_ms,0,blend_radius_m)
    |   movel([0.528500, -1.441980, -2.531312, -0.739098, 1.570796, 2.099296],accel_mss,speed_ms,0,blend_radius_m)
    |   movel([0.528712, -1.441319, -2.531837, -0.739233, 1.570796, 2.099508],accel_mss,speed_ms,0,blend_radius_m)
    |   movel([0.528754, -1.440900, -2.532170, -0.739319, 1.570796, 2.099550],accel_mss,speed_ms,0,blend_radius_m)
    |   movel([0.528518, -1.440358, -2.532599, -0.739431, 1.570796, 2.099315],accel_mss,speed_ms,0,blend_radius_m)
    |   movel([0.528131, -1.440101, -2.532804, -0.739485, 1.570796, 2.098927],accel_mss,speed_ms,0,blend_radius_m)
    |   movel([0.527622, -1.440071, -2.532827, -0.739491, 1.570796, 2.098419],accel_mss,speed_ms,0,blend_radius_m)
    |   movel([0.527024, -1.440220, -2.532709, -0.739460, 1.570796, 2.097821],accel_mss,speed_ms,0,blend_radius_m)
    |   movel([0.525708, -1.440829, -2.532226, -0.739334, 1.570796, 2.096504],accel_mss,speed_ms,0,blend_radius_m)
    |   movel([0.524451, -1.441503, -2.531691, -0.739195, 1.570796, 2.095247],accel_mss,speed_ms,0,blend_radius_m)
    |   movel([0.522478, -1.442423, -2.530959, -0.739007, 1.570796, 2.093274],accel_mss,speed_ms,0,blend_radius_m)
    |   movel([0.520576, -1.443144, -2.530385, -0.738861, 1.570796, 2.091372],accel_mss,speed_ms,0,blend_radius_m)
    |   movel([0.518692, -1.443593, -2.530026, -0.738770, 1.570796, 2.089489],accel_mss,speed_ms,0,blend_radius_m)
    |   movel([0.516787, -1.443689, -2.529949, -0.738750, 1.570796, 2.087583],accel_mss,speed_ms,0,blend_radius_m)
    |   movel([0.518245, -1.442894, -2.530584, -0.738911, 1.570796, 2.089042],accel_mss,speed_ms,0,blend_radius_m)
    |   movel([0.519593, -1.441927, -2.531353, -0.739108, 1.570796, 2.090389],accel_mss,speed_ms,0,blend_radius_m)
    |   movel([0.520169, -1.441329, -2.531829, -0.739231, 1.570796, 2.090965],accel_mss,speed_ms,0,blend_radius_m)
    |   movel([0.520610, -1.440680, -2.532344, -0.739365, 1.570796, 2.091406],accel_mss,speed_ms,0,blend_radius_m)
    |   movel([0.520870, -1.440025, -2.532863, -0.739500, 1.570796, 2.091666],accel_mss,speed_ms,0,blend_radius_m)
    |   movel([0.520888, -1.439417, -2.533345, -0.739627, 1.570796, 2.091684],accel_mss,speed_ms,0,blend_radius_m)
    |   movel([0.520543, -1.438832, -2.533808, -0.739749, 1.570796, 2.091340],accel_mss,speed_ms,0,blend_radius_m)
    |   movel([0.519903, -1.438483, -2.534084, -0.739822, 1.570796, 2.090700],accel_mss,speed_ms,0,blend_radius_m)
    |   movel([0.519080, -1.438310, -2.534221, -0.739858, 1.570796, 2.089876],accel_mss,speed_ms,0,blend_radius_m)
    |   movel([0.518194, -1.438247, -2.534271, -0.739872, 1.570796, 2.088990],accel_mss,speed_ms,0,blend_radius_m)
    |   speed_ms = 0.005
    |   movel([0.518194, -1.429866, -2.530530, -0.751993, 1.570796, 2.088990],accel_mss,speed_ms,0,blend_radius_m)
    |   speed_ms = 0.040
    |   movel([0.510141, -1.449455, -2.514970, -0.747963, 1.570796, 2.080938],accel_mss,speed_ms,0,blend_radius_m)
    |   speed_ms = 0.005
    |   movel([0.510141, -1.457684, -2.518629, -0.736076, 1.570796, 2.080938],accel_mss,speed_ms,0,blend_radius_m)
    |   speed_ms = 0.025
    |   movel([0.511091, -1.456693, -2.519440, -0.736256, 1.570796, 2.081888],accel_mss,speed_ms,0,blend_radius_m)
    |   movel([0.512141, -1.455770, -2.520195, -0.736424, 1.570796, 2.082937],accel_mss,speed_ms,0,blend_radius_m)
    |   movel([0.513267, -1.454927, -2.520883, -0.736579, 1.570796, 2.084063],accel_mss,speed_ms,0,blend_radius_m)
    |   movel([0.514457, -1.454175, -2.521496, -0.736718, 1.570796, 2.085253],accel_mss,speed_ms,0,blend_radius_m)
    |   movel([0.515692, -1.453521, -2.522028, -0.736840, 1.570796, 2.086488],accel_mss,speed_ms,0,blend_radius_m)
    |   movel([0.516954, -1.452980, -2.522467, -0.736941, 1.570796, 2.087750],accel_mss,speed_ms,0,blend_radius_m)
    |   movel([0.518224, -1.452560, -2.522808, -0.737020, 1.570796, 2.089020],accel_mss,speed_ms,0,blend_radius_m)
    |   movel([0.519487, -1.452271, -2.523043, -0.737075, 1.570796, 2.090284],accel_mss,speed_ms,0,blend_radius_m)
    |   movel([0.521308, -1.452078, -2.523200, -0.737111, 1.570796, 2.092104],accel_mss,speed_ms,0,blend_radius_m)
    |   movel([0.522944, -1.452159, -2.523134, -0.737096, 1.570796, 2.093740],accel_mss,speed_ms,0,blend_radius_m)
    |   movel([0.524404, -1.452488, -2.522867, -0.737034, 1.570796, 2.095200],accel_mss,speed_ms,0,blend_radius_m)
    |   movel([0.525694, -1.453041, -2.522418, -0.736930, 1.570796, 2.096491],accel_mss,speed_ms,0,blend_radius_m)
    |   movel([0.526823, -1.453792, -2.521807, -0.736790, 1.570796, 2.097619],accel_mss,speed_ms,0,blend_radius_m)
    |   movel([0.527798, -1.454719, -2.521052, -0.736618, 1.570796, 2.098594],accel_mss,speed_ms,0,blend_radius_m)
    |   movel([0.528624, -1.455797, -2.520173, -0.736419, 1.570796, 2.099421],accel_mss,speed_ms,0,blend_radius_m)
    |   movel([0.529313, -1.457000, -2.519189, -0.736200, 1.570796, 2.100109],accel_mss,speed_ms,0,blend_radius_m)
    |   movel([0.529870, -1.458305, -2.518119, -0.735965, 1.570796, 2.100667],accel_mss,speed_ms,0,blend_radius_m)
    |   movel([0.530307, -1.459689, -2.516982, -0.735718, 1.570796, 2.101103],accel_mss,speed_ms,0,blend_radius_m)
    |   movel([0.530848, -1.462592, -2.514587, -0.735210, 1.570796, 2.101644],accel_mss,speed_ms,0,blend_radius_m)
    |   movel([0.531006, -1.465517, -2.512160, -0.734712, 1.570796, 2.101803],accel_mss,speed_ms,0,blend_radius_m)
    |   movel([0.530842, -1.468282, -2.509854, -0.734253, 1.570796, 2.101639],accel_mss,speed_ms,0,blend_radius_m)
    |   movel([0.530390, -1.471193, -2.507413, -0.733783, 1.570796, 2.101186],accel_mss,speed_ms,0,blend_radius_m)
    |   movel([0.529720, -1.474131, -2.504936, -0.733322, 1.570796, 2.100516],accel_mss,speed_ms,0,blend_radius_m)
    |   movel([0.528861, -1.477086, -2.502431, -0.732872, 1.570796, 2.099658],accel_mss,speed_ms,0,blend_radius_m)
    |   movel([0.527841, -1.480049, -2.499906, -0.732435, 1.570796, 2.098637],accel_mss,speed_ms,0,blend_radius_m)
    |   movel([0.526687, -1.483008, -2.497369, -0.732012, 1.570796, 2.097483],accel_mss,speed_ms,0,blend_radius_m)
    |   movel([0.525429, -1.485956, -2.494829, -0.731604, 1.570796, 2.096225],accel_mss,speed_ms,0,blend_radius_m)
    |   movel([0.522707, -1.491776, -2.489774, -0.730839, 1.570796, 2.093504],accel_mss,speed_ms,0,blend_radius_m)
    |   movel([0.520789, -1.495817, -2.486233, -0.730340, 1.570796, 2.091586],accel_mss,speed_ms,0,blend_radius_m)
    |   movel([0.519999, -1.497823, -2.484465, -0.730101, 1.570796, 2.090795],accel_mss,speed_ms,0,blend_radius_m)
    |   movel([0.519432, -1.499808, -2.482709, -0.729872, 1.570796, 2.090228],accel_mss,speed_ms,0,blend_radius_m)
    |   movel([0.519026, -1.502378, -2.480427, -0.729584, 1.570796, 2.089822],accel_mss,speed_ms,0,blend_radius_m)
    |   movel([0.518624, -1.504952, -2.478131, -0.729306, 1.570796, 2.089420],accel_mss,speed_ms,0,blend_radius_m)
    |   movel([0.518292, -1.506214, -2.477001, -0.729174, 1.570796, 2.089088],accel_mss,speed_ms,0,blend_radius_m)
    |   movel([0.517800, -1.507448, -2.475895, -0.729047, 1.570796, 2.088596],accel_mss,speed_ms,0,blend_radius_m)
    |   movel([0.517098, -1.508640, -2.474823, -0.728926, 1.570796, 2.087894],accel_mss,speed_ms,0,blend_radius_m)
    |   movel([0.516134, -1.509785, -2.473791, -0.728813, 1.570796, 2.086930],accel_mss,speed_ms,0,blend_radius_m)
    |   movel([0.518755, -1.507097, -2.476210, -0.729083, 1.570796, 2.089552],accel_mss,speed_ms,0,blend_radius_m)
    |   movel([0.521247, -1.504345, -2.478673, -0.729371, 1.570796, 2.092043],accel_mss,speed_ms,0,blend_radius_m)
    |   movel([0.526020, -1.498683, -2.483705, -0.730001, 1.570796, 2.096816],accel_mss,speed_ms,0,blend_radius_m)
    |   movel([0.528599, -1.495468, -2.486539, -0.730382, 1.570796, 2.099395],accel_mss,speed_ms,0,blend_radius_m)
    |   movel([0.531106, -1.492207, -2.489397, -0.730784, 1.570796, 2.101903],accel_mss,speed_ms,0,blend_radius_m)
    |   movel([0.535966, -1.485569, -2.495163, -0.731657, 1.570796, 2.106762],accel_mss,speed_ms,0,blend_radius_m)
    |   movel([0.540563, -1.478943, -2.500850, -0.732596, 1.570796, 2.111359],accel_mss,speed_ms,0,blend_radius_m)
    |   movel([0.542732, -1.475555, -2.503731, -0.733104, 1.570796, 2.113528],accel_mss,speed_ms,0,blend_radius_m)
    |   movel([0.544723, -1.472142, -2.506614, -0.733633, 1.570796, 2.115519],accel_mss,speed_ms,0,blend_radius_m)
    |   movel([0.546112, -1.469422, -2.508900, -0.734068, 1.570796, 2.116908],accel_mss,speed_ms,0,blend_radius_m)
    |   movel([0.547394, -1.466668, -2.511201, -0.734519, 1.570796, 2.118190],accel_mss,speed_ms,0,blend_radius_m)
    |   movel([0.548701, -1.463889, -2.513512, -0.734988, 1.570796, 2.119497],accel_mss,speed_ms,0,blend_radius_m)
    |   movel([0.550164, -1.461093, -2.515825, -0.735471, 1.570796, 2.120961],accel_mss,speed_ms,0,blend_radius_m)
    |   movel([0.550637, -1.460364, -2.516426, -0.735599, 1.570796, 2.121434],accel_mss,speed_ms,0,blend_radius_m)
    |   movel([0.551236, -1.459675, -2.516993, -0.735720, 1.570796, 2.122032],accel_mss,speed_ms,0,blend_radius_m)
    |   movel([0.551916, -1.459170, -2.517409, -0.735810, 1.570796, 2.122713],accel_mss,speed_ms,0,blend_radius_m)
    |   movel([0.552279, -1.459029, -2.517525, -0.735835, 1.570796, 2.123075],accel_mss,speed_ms,0,blend_radius_m)
    |   movel([0.552650, -1.458984, -2.517562, -0.735843, 1.570796, 2.123447],accel_mss,speed_ms,0,blend_radius_m)
    |   movel([0.553094, -1.459095, -2.517470, -0.735823, 1.570796, 2.123890],accel_mss,speed_ms,0,blend_radius_m)
    |   movel([0.553450, -1.459322, -2.517284, -0.735783, 1.570796, 2.124247],accel_mss,speed_ms,0,blend_radius_m)
    |   movel([0.555162, -1.460824, -2.516047, -0.735518, 1.570796, 2.125958],accel_mss,speed_ms,0,blend_radius_m)
    |   movel([0.556530, -1.462499, -2.514664, -0.735226, 1.570796, 2.127326],accel_mss,speed_ms,0,blend_radius_m)
    |   movel([0.557585, -1.464326, -2.513150, -0.734913, 1.570796, 2.128381],accel_mss,speed_ms,0,blend_radius_m)
    |   movel([0.558352, -1.466294, -2.511513, -0.734582, 1.570796, 2.129148],accel_mss,speed_ms,0,blend_radius_m)
    |   movel([0.558858, -1.468380, -2.509772, -0.734237, 1.570796, 2.129655],accel_mss,speed_ms,0,blend_radius_m)
    |   movel([0.559133, -1.470569, -2.507937, -0.733883, 1.570796, 2.129930],accel_mss,speed_ms,0,blend_radius_m)
    |   movel([0.559203, -1.472844, -2.506022, -0.733522, 1.570796, 2.129999],accel_mss,speed_ms,0,blend_radius_m)
    |   movel([0.559091, -1.475191, -2.504039, -0.733159, 1.570796, 2.129888],accel_mss,speed_ms,0,blend_radius_m)
    |   movel([0.558827, -1.477592, -2.502001, -0.732796, 1.570796, 2.129624],accel_mss,speed_ms,0,blend_radius_m)
    |   movel([0.558438, -1.480032, -2.499920, -0.732437, 1.570796, 2.129235],accel_mss,speed_ms,0,blend_radius_m)
    |   movel([0.557386, -1.484964, -2.495685, -0.731739, 1.570796, 2.128183],accel_mss,speed_ms,0,blend_radius_m)
    |   movel([0.554892, -1.494646, -2.487262, -0.730482, 1.570796, 2.125689],accel_mss,speed_ms,0,blend_radius_m)
    |   movel([0.554588, -1.496145, -2.485944, -0.730300, 1.570796, 2.125384],accel_mss,speed_ms,0,blend_radius_m)
    |   movel([0.554575, -1.496851, -2.485322, -0.730216, 1.570796, 2.125371],accel_mss,speed_ms,0,blend_radius_m)
    |   movel([0.554722, -1.497492, -2.484757, -0.730140, 1.570796, 2.125519],accel_mss,speed_ms,0,blend_radius_m)
    |   movel([0.555275, -1.498243, -2.484094, -0.730052, 1.570796, 2.126071],accel_mss,speed_ms,0,blend_radius_m)
    |   movel([0.555655, -1.498482, -2.483883, -0.730024, 1.570796, 2.126451],accel_mss,speed_ms,0,blend_radius_m)
    |   movel([0.556095, -1.498637, -2.483746, -0.730006, 1.570796, 2.126891],accel_mss,speed_ms,0,blend_radius_m)
    |   movel([0.557113, -1.498726, -2.483667, -0.729996, 1.570796, 2.127910],accel_mss,speed_ms,0,blend_radius_m)
    |   movel([0.558266, -1.498560, -2.483813, -0.730015, 1.570796, 2.129063],accel_mss,speed_ms,0,blend_radius_m)
    |   movel([0.559484, -1.498195, -2.484136, -0.730058, 1.570796, 2.130280],accel_mss,speed_ms,0,blend_radius_m)
    |   movel([0.560700, -1.497680, -2.484591, -0.730118, 1.570796, 2.131496],accel_mss,speed_ms,0,blend_radius_m)
    |   movel([0.561849, -1.497066, -2.485132, -0.730190, 1.570796, 2.132646],accel_mss,speed_ms,0,blend_radius_m)
    |   movel([0.562859, -1.496403, -2.485717, -0.730269, 1.570796, 2.133656],accel_mss,speed_ms,0,blend_radius_m)
    |   movel([0.564501, -1.495161, -2.486809, -0.730419, 1.570796, 2.135297],accel_mss,speed_ms,0,blend_radius_m)
    |   movel([0.566103, -1.493854, -2.487956, -0.730579, 1.570796, 2.136900],accel_mss,speed_ms,0,blend_radius_m)
    |   movel([0.569169, -1.491072, -2.490389, -0.730929, 1.570796, 2.139965],accel_mss,speed_ms,0,blend_radius_m)
    |   movel([0.572027, -1.488119, -2.492957, -0.731313, 1.570796, 2.142824],accel_mss,speed_ms,0,blend_radius_m)
    |   movel([0.574646, -1.485054, -2.495608, -0.731727, 1.570796, 2.145443],accel_mss,speed_ms,0,blend_radius_m)
    |   movel([0.575591, -1.483880, -2.496620, -0.731890, 1.570796, 2.146387],accel_mss,speed_ms,0,blend_radius_m)
    |   movel([0.576618, -1.482762, -2.497581, -0.732046, 1.570796, 2.147414],accel_mss,speed_ms,0,blend_radius_m)
    |   movel([0.577188, -1.482268, -2.498005, -0.732116, 1.570796, 2.147985],accel_mss,speed_ms,0,blend_radius_m)
    |   movel([0.577814, -1.481835, -2.498377, -0.732178, 1.570796, 2.148610],accel_mss,speed_ms,0,blend_radius_m)
    |   movel([0.578503, -1.481482, -2.498679, -0.732228, 1.570796, 2.149299],accel_mss,speed_ms,0,blend_radius_m)
    |   movel([0.579266, -1.481229, -2.498896, -0.732264, 1.570796, 2.150062],accel_mss,speed_ms,0,blend_radius_m)
    |   movel([0.580251, -1.481159, -2.498956, -0.732274, 1.570796, 2.151047],accel_mss,speed_ms,0,blend_radius_m)
    |   movel([0.581073, -1.481422, -2.498731, -0.732237, 1.570796, 2.151869],accel_mss,speed_ms,0,blend_radius_m)
    |   movel([0.581707, -1.481932, -2.498293, -0.732164, 1.570796, 2.152503],accel_mss,speed_ms,0,blend_radius_m)
    |   movel([0.582136, -1.482605, -2.497715, -0.732068, 1.570796, 2.152933],accel_mss,speed_ms,0,blend_radius_m)
    |   movel([0.582578, -1.483885, -2.496615, -0.731889, 1.570796, 2.153374],accel_mss,speed_ms,0,blend_radius_m)
    |   movel([0.582850, -1.485265, -2.495426, -0.731698, 1.570796, 2.153646],accel_mss,speed_ms,0,blend_radius_m)
    |   movel([0.583065, -1.488131, -2.492947, -0.731312, 1.570796, 2.153861],accel_mss,speed_ms,0,blend_radius_m)
    |   movel([0.583037, -1.489513, -2.491746, -0.731130, 1.570796, 2.153834],accel_mss,speed_ms,0,blend_radius_m)
    |   movel([0.582882, -1.490891, -2.490546, -0.730952, 1.570796, 2.153679],accel_mss,speed_ms,0,blend_radius_m)
    |   movel([0.582611, -1.492261, -2.489350, -0.730778, 1.570796, 2.153407],accel_mss,speed_ms,0,blend_radius_m)
    |   movel([0.582227, -1.493625, -2.488157, -0.730607, 1.570796, 2.153023],accel_mss,speed_ms,0,blend_radius_m)
    |   movel([0.581738, -1.494980, -2.486969, -0.730441, 1.570796, 2.152535],accel_mss,speed_ms,0,blend_radius_m)
    |   movel([0.580473, -1.497665, -2.484604, -0.730120, 1.570796, 2.151270],accel_mss,speed_ms,0,blend_radius_m)
    |   movel([0.579710, -1.498992, -2.483432, -0.729965, 1.570796, 2.150506],accel_mss,speed_ms,0,blend_radius_m)
    |   movel([0.577960, -1.501613, -2.481108, -0.729668, 1.570796, 2.148756],accel_mss,speed_ms,0,blend_radius_m)
    |   movel([0.575952, -1.504185, -2.478816, -0.729388, 1.570796, 2.146749],accel_mss,speed_ms,0,blend_radius_m)
    |   movel([0.573737, -1.506705, -2.476561, -0.729123, 1.570796, 2.144533],accel_mss,speed_ms,0,blend_radius_m)
    |   movel([0.571371, -1.509163, -2.474352, -0.728874, 1.570796, 2.142167],accel_mss,speed_ms,0,blend_radius_m)
    |   movel([0.567732, -1.512631, -2.471218, -0.728540, 1.570796, 2.138528],accel_mss,speed_ms,0,blend_radius_m)
    |   movel([0.565824, -1.514296, -2.469707, -0.728386, 1.570796, 2.136621],accel_mss,speed_ms,0,blend_radius_m)
    |   movel([0.563854, -1.515893, -2.468253, -0.728243, 1.570796, 2.134651],accel_mss,speed_ms,0,blend_radius_m)
    |   movel([0.561822, -1.517401, -2.466876, -0.728112, 1.570796, 2.132618],accel_mss,speed_ms,0,blend_radius_m)
    |   movel([0.559727, -1.518806, -2.465590, -0.727992, 1.570796, 2.130523],accel_mss,speed_ms,0,blend_radius_m)
    |   movel([0.557561, -1.520091, -2.464412, -0.727886, 1.570796, 2.128357],accel_mss,speed_ms,0,blend_radius_m)
    |   movel([0.555327, -1.521236, -2.463359, -0.727794, 1.570796, 2.126124],accel_mss,speed_ms,0,blend_radius_m)
    |   movel([0.552124, -1.522621, -2.462084, -0.727685, 1.570796, 2.122920],accel_mss,speed_ms,0,blend_radius_m)
    |   movel([0.550419, -1.523230, -2.461521, -0.727638, 1.570796, 2.121215],accel_mss,speed_ms,0,blend_radius_m)
    |   movel([0.548705, -1.523722, -2.461067, -0.727600, 1.570796, 2.119502],accel_mss,speed_ms,0,blend_radius_m)
    |   movel([0.547032, -1.524050, -2.460764, -0.727575, 1.570796, 2.117828],accel_mss,speed_ms,0,blend_radius_m)
    |   movel([0.545444, -1.524166, -2.460656, -0.727567, 1.570796, 2.116240],accel_mss,speed_ms,0,blend_radius_m)
    |   movel([0.543989, -1.524022, -2.460790, -0.727577, 1.570796, 2.114785],accel_mss,speed_ms,0,blend_radius_m)
    |   movel([0.543326, -1.523839, -2.460959, -0.727591, 1.570796, 2.114122],accel_mss,speed_ms,0,blend_radius_m)
    |   movel([0.542715, -1.523572, -2.461206, -0.727611, 1.570796, 2.113512],accel_mss,speed_ms,0,blend_radius_m)
    |   movel([0.542106, -1.523172, -2.461575, -0.727642, 1.570796, 2.112902],accel_mss,speed_ms,0,blend_radius_m)
    |   movel([0.541607, -1.522687, -2.462022, -0.727679, 1.570796, 2.112403],accel_mss,speed_ms,0,blend_radius_m)
    |   movel([0.541207, -1.522126, -2.462540, -0.727723, 1.570796, 2.112004],accel_mss,speed_ms,0,blend_radius_m)
    |   movel([0.540902, -1.521496, -2.463120, -0.727773, 1.570796, 2.111698],accel_mss,speed_ms,0,blend_radius_m)
    |   movel([0.540535, -1.520068, -2.464433, -0.727888, 1.570796, 2.111331],accel_mss,speed_ms,0,blend_radius_m)
    |   movel([0.540444, -1.518473, -2.465896, -0.728020, 1.570796, 2.111240],accel_mss,speed_ms,0,blend_radius_m)
    |   movel([0.540559, -1.516785, -2.467439, -0.728165, 1.570796, 2.111355],accel_mss,speed_ms,0,blend_radius_m)
    |   movel([0.540816, -1.515077, -2.468996, -0.728316, 1.570796, 2.111612],accel_mss,speed_ms,0,blend_radius_m)
    |   movel([0.541487, -1.511892, -2.471888, -0.728610, 1.570796, 2.112284],accel_mss,speed_ms,0,blend_radius_m)
    |   movel([0.541819, -1.510404, -2.473232, -0.728752, 1.570796, 2.112615],accel_mss,speed_ms,0,blend_radius_m)
    |   movel([0.541998, -1.508958, -2.474537, -0.728895, 1.570796, 2.112794],accel_mss,speed_ms,0,blend_radius_m)
    |   movel([0.541952, -1.508290, -2.475137, -0.728961, 1.570796, 2.112748],accel_mss,speed_ms,0,blend_radius_m)
    |   movel([0.541774, -1.507681, -2.475685, -0.729023, 1.570796, 2.112571],accel_mss,speed_ms,0,blend_radius_m)
    |   movel([0.541434, -1.507148, -2.476163, -0.729077, 1.570796, 2.112230],accel_mss,speed_ms,0,blend_radius_m)
    |   movel([0.540901, -1.506706, -2.476560, -0.729123, 1.570796, 2.111697],accel_mss,speed_ms,0,blend_radius_m)
    |   movel([0.540999, -1.506837, -2.476443, -0.729109, 1.570796, 2.111796],accel_mss,speed_ms,0,blend_radius_m)
    |   movel([0.540993, -1.507039, -2.476261, -0.729088, 1.570796, 2.111789],accel_mss,speed_ms,0,blend_radius_m)
    |   movel([0.540687, -1.507637, -2.475725, -0.729027, 1.570796, 2.111483],accel_mss,speed_ms,0,blend_radius_m)
    |   movel([0.540031, -1.508460, -2.474985, -0.728944, 1.570796, 2.110827],accel_mss,speed_ms,0,blend_radius_m)
    |   movel([0.539081, -1.509472, -2.474073, -0.728844, 1.570796, 2.109877],accel_mss,speed_ms,0,blend_radius_m)
    |   movel([0.536506, -1.511911, -2.471870, -0.728608, 1.570796, 2.107302],accel_mss,speed_ms,0,blend_radius_m)
    |   movel([0.533377, -1.514652, -2.469383, -0.728354, 1.570796, 2.104174],accel_mss,speed_ms,0,blend_radius_m)
    |   movel([0.527088, -1.519857, -2.464627, -0.727905, 1.570796, 2.097884],accel_mss,speed_ms,0,blend_radius_m)
    |   movel([0.523408, -1.522733, -2.461980, -0.727676, 1.570796, 2.094204],accel_mss,speed_ms,0,blend_radius_m)
    |   movel([0.519372, -1.525494, -2.459426, -0.727468, 1.570796, 2.090168],accel_mss,speed_ms,0,blend_radius_m)
    |   movel([0.515337, -1.528147, -2.456962, -0.727280, 1.570796, 2.086134],accel_mss,speed_ms,0,blend_radius_m)
    |   movel([0.511276, -1.530728, -2.454553, -0.727108, 1.570796, 2.082072],accel_mss,speed_ms,0,blend_radius_m)
    |   movel([0.503302, -1.535575, -2.450000, -0.726814, 1.570796, 2.074098],accel_mss,speed_ms,0,blend_radius_m)
    |   movel([0.499392, -1.537721, -2.447972, -0.726695, 1.570796, 2.070188],accel_mss,speed_ms,0,blend_radius_m)
    |   movel([0.497416, -1.538674, -2.447070, -0.726645, 1.570796, 2.068213],accel_mss,speed_ms,0,blend_radius_m)
    |   movel([0.495430, -1.539517, -2.446269, -0.726602, 1.570796, 2.066226],accel_mss,speed_ms,0,blend_radius_m)
    |   movel([0.493429, -1.540226, -2.445596, -0.726567, 1.570796, 2.064225],accel_mss,speed_ms,0,blend_radius_m)
    |   movel([0.491417, -1.540779, -2.445070, -0.726540, 1.570796, 2.062214],accel_mss,speed_ms,0,blend_radius_m)
    |   movel([0.493294, -1.537726, -2.447968, -0.726695, 1.570796, 2.064090],accel_mss,speed_ms,0,blend_radius_m)
    |   movel([0.493731, -1.536801, -2.448843, -0.726745, 1.570796, 2.064527],accel_mss,speed_ms,0,blend_radius_m)
    |   movel([0.493771, -1.536384, -2.449237, -0.726768, 1.570796, 2.064567],accel_mss,speed_ms,0,blend_radius_m)
    |   movel([0.493597, -1.536066, -2.449537, -0.726786, 1.570796, 2.064394],accel_mss,speed_ms,0,blend_radius_m)
    |   movel([0.493297, -1.535935, -2.449661, -0.726793, 1.570796, 2.064093],accel_mss,speed_ms,0,blend_radius_m)
    |   movel([0.492915, -1.535922, -2.449673, -0.726794, 1.570796, 2.063711],accel_mss,speed_ms,0,blend_radius_m)
    |   movel([0.490914, -1.536231, -2.449382, -0.726777, 1.570796, 2.061711],accel_mss,speed_ms,0,blend_radius_m)
    |   movel([0.489818, -1.536232, -2.449381, -0.726777, 1.570796, 2.060615],accel_mss,speed_ms,0,blend_radius_m)
    |   movel([0.488797, -1.536075, -2.449529, -0.726785, 1.570796, 2.059594],accel_mss,speed_ms,0,blend_radius_m)
    |   movel([0.487879, -1.535763, -2.449823, -0.726803, 1.570796, 2.058675],accel_mss,speed_ms,0,blend_radius_m)
    |   movel([0.487648, -1.535578, -2.449998, -0.726813, 1.570796, 2.058445],accel_mss,speed_ms,0,blend_radius_m)
    |   movel([0.487677, -1.535333, -2.450228, -0.726827, 1.570796, 2.058473],accel_mss,speed_ms,0,blend_radius_m)
    |   movel([0.488374, -1.534524, -2.450991, -0.726874, 1.570796, 2.059170],accel_mss,speed_ms,0,blend_radius_m)
    |   movel([0.488495, -1.534216, -2.451281, -0.726892, 1.570796, 2.059291],accel_mss,speed_ms,0,blend_radius_m)
    |   movel([0.488458, -1.533935, -2.451545, -0.726909, 1.570796, 2.059254],accel_mss,speed_ms,0,blend_radius_m)
    |   movel([0.488296, -1.533709, -2.451758, -0.726922, 1.570796, 2.059092],accel_mss,speed_ms,0,blend_radius_m)
    |   movel([0.488039, -1.533564, -2.451894, -0.726931, 1.570796, 2.058835],accel_mss,speed_ms,0,blend_radius_m)
    |   movel([0.487372, -1.533509, -2.451945, -0.726934, 1.570796, 2.058169],accel_mss,speed_ms,0,blend_radius_m)
    |   movel([0.482012, -1.534472, -2.451040, -0.726877, 1.570796, 2.052809],accel_mss,speed_ms,0,blend_radius_m)
    |   movel([0.483729, -1.533917, -2.451562, -0.726910, 1.570796, 2.054525],accel_mss,speed_ms,0,blend_radius_m)
    |   movel([0.485480, -1.533241, -2.452198, -0.726951, 1.570796, 2.056276],accel_mss,speed_ms,0,blend_radius_m)
    |   movel([0.487243, -1.532463, -2.452928, -0.726998, 1.570796, 2.058040],accel_mss,speed_ms,0,blend_radius_m)
    |   movel([0.489007, -1.531599, -2.453738, -0.727052, 1.570796, 2.059803],accel_mss,speed_ms,0,blend_radius_m)
    |   movel([0.492467, -1.529679, -2.455534, -0.727177, 1.570796, 2.063264],accel_mss,speed_ms,0,blend_radius_m)
    |   movel([0.495725, -1.527617, -2.457455, -0.727317, 1.570796, 2.066521],accel_mss,speed_ms,0,blend_radius_m)
    |   movel([0.499158, -1.525260, -2.459643, -0.727485, 1.570796, 2.069954],accel_mss,speed_ms,0,blend_radius_m)
    |   movel([0.502533, -1.522773, -2.461943, -0.727673, 1.570796, 2.073330],accel_mss,speed_ms,0,blend_radius_m)
    |   movel([0.504170, -1.521467, -2.463147, -0.727775, 1.570796, 2.074966],accel_mss,speed_ms,0,blend_radius_m)
    |   movel([0.505759, -1.520115, -2.464390, -0.727884, 1.570796, 2.076556],accel_mss,speed_ms,0,blend_radius_m)
    |   movel([0.507286, -1.518712, -2.465677, -0.728000, 1.570796, 2.078082],accel_mss,speed_ms,0,blend_radius_m)
    |   movel([0.508742, -1.517249, -2.467015, -0.728125, 1.570796, 2.079538],accel_mss,speed_ms,0,blend_radius_m)
    |   movel([0.509588, -1.516300, -2.467881, -0.728207, 1.570796, 2.080384],accel_mss,speed_ms,0,blend_radius_m)
    |   movel([0.510366, -1.515308, -2.468786, -0.728295, 1.570796, 2.081163],accel_mss,speed_ms,0,blend_radius_m)
    |   movel([0.511731, -1.513219, -2.470684, -0.728485, 1.570796, 2.082527],accel_mss,speed_ms,0,blend_radius_m)
    |   movel([0.512844, -1.511031, -2.472666, -0.728692, 1.570796, 2.083641],accel_mss,speed_ms,0,blend_radius_m)
    |   movel([0.513716, -1.508789, -2.474689, -0.728912, 1.570796, 2.084513],accel_mss,speed_ms,0,blend_radius_m)
    |   movel([0.514362, -1.506538, -2.476711, -0.729140, 1.570796, 2.085158],accel_mss,speed_ms,0,blend_radius_m)
    |   movel([0.514791, -1.504328, -2.478688, -0.729372, 1.570796, 2.085588],accel_mss,speed_ms,0,blend_radius_m)
    |   movel([0.515013, -1.502206, -2.480580, -0.729603, 1.570796, 2.085809],accel_mss,speed_ms,0,blend_radius_m)
    |   movel([0.515040, -1.500220, -2.482344, -0.729825, 1.570796, 2.085836],accel_mss,speed_ms,0,blend_radius_m)
    |   movel([0.514833, -1.499178, -2.483268, -0.729944, 1.570796, 2.085629],accel_mss,speed_ms,0,blend_radius_m)
    |   movel([0.514328, -1.498388, -2.483965, -0.730035, 1.570796, 2.085125],accel_mss,speed_ms,0,blend_radius_m)
    |   movel([0.513576, -1.497861, -2.484431, -0.730097, 1.570796, 2.084372],accel_mss,speed_ms,0,blend_radius_m)
    |   movel([0.512626, -1.497606, -2.484656, -0.730127, 1.570796, 2.083422],accel_mss,speed_ms,0,blend_radius_m)
    |   movel([0.511527, -1.497627, -2.484638, -0.730124, 1.570796, 2.082323],accel_mss,speed_ms,0,blend_radius_m)
    |   movel([0.510328, -1.497933, -2.484368, -0.730088, 1.570796, 2.081125],accel_mss,speed_ms,0,blend_radius_m)
    |   movel([0.509087, -1.498529, -2.483841, -0.730019, 1.570796, 2.079883],accel_mss,speed_ms,0,blend_radius_m)
    |   movel([0.507849, -1.499420, -2.483053, -0.729916, 1.570796, 2.078646],accel_mss,speed_ms,0,blend_radius_m)
    |   movel([0.506057, -1.500901, -2.481740, -0.729748, 1.570796, 2.076853],accel_mss,speed_ms,0,blend_radius_m)
    |   movel([0.504215, -1.502308, -2.480490, -0.729592, 1.570796, 2.075011],accel_mss,speed_ms,0,blend_radius_m)
    |   movel([0.502327, -1.503615, -2.479325, -0.729449, 1.570796, 2.073123],accel_mss,speed_ms,0,blend_radius_m)
    |   movel([0.500388, -1.504800, -2.478267, -0.729322, 1.570796, 2.071184],accel_mss,speed_ms,0,blend_radius_m)
    |   movel([0.498404, -1.505837, -2.477339, -0.729213, 1.570796, 2.069200],accel_mss,speed_ms,0,blend_radius_m)
    |   movel([0.496371, -1.506704, -2.476562, -0.729123, 1.570796, 2.067167],accel_mss,speed_ms,0,blend_radius_m)
    |   movel([0.494289, -1.507378, -2.475957, -0.729054, 1.570796, 2.065085],accel_mss,speed_ms,0,blend_radius_m)
    |   movel([0.492160, -1.507833, -2.475548, -0.729008, 1.570796, 2.062956],accel_mss,speed_ms,0,blend_radius_m)
    |   movel([0.491077, -1.507930, -2.475462, -0.728998, 1.570796, 2.061873],accel_mss,speed_ms,0,blend_radius_m)
    |   movel([0.490044, -1.507891, -2.475496, -0.729002, 1.570796, 2.060840],accel_mss,speed_ms,0,blend_radius_m)
    |   movel([0.488081, -1.507580, -2.475776, -0.729033, 1.570796, 2.058877],accel_mss,speed_ms,0,blend_radius_m)
    |   movel([0.486632, -1.507175, -2.476139, -0.729075, 1.570796, 2.057428],accel_mss,speed_ms,0,blend_radius_m)
    |   movel([0.485361, -1.506589, -2.476665, -0.729135, 1.570796, 2.056158],accel_mss,speed_ms,0,blend_radius_m)
    |   movel([0.484262, -1.505838, -2.477338, -0.729213, 1.570796, 2.055058],accel_mss,speed_ms,0,blend_radius_m)
    |   movel([0.483321, -1.504938, -2.478144, -0.729308, 1.570796, 2.054117],accel_mss,speed_ms,0,blend_radius_m)
    |   movel([0.482527, -1.503906, -2.479066, -0.729418, 1.570796, 2.053323],accel_mss,speed_ms,0,blend_radius_m)
    |   movel([0.481869, -1.502756, -2.480091, -0.729542, 1.570796, 2.052665],accel_mss,speed_ms,0,blend_radius_m)
    |   movel([0.481342, -1.501504, -2.481204, -0.729680, 1.570796, 2.052138],accel_mss,speed_ms,0,blend_radius_m)
    |   movel([0.480931, -1.500169, -2.482389, -0.729831, 1.570796, 2.051727],accel_mss,speed_ms,0,blend_radius_m)
    |   movel([0.480626, -1.498766, -2.483631, -0.729991, 1.570796, 2.051422],accel_mss,speed_ms,0,blend_radius_m)
    |   movel([0.480420, -1.497308, -2.484919, -0.730162, 1.570796, 2.051216],accel_mss,speed_ms,0,blend_radius_m)
    |   movel([0.480258, -1.494306, -2.487560, -0.730523, 1.570796, 2.051054],accel_mss,speed_ms,0,blend_radius_m)
    |   movel([0.480362, -1.491291, -2.490197, -0.730901, 1.570796, 2.051158],accel_mss,speed_ms,0,blend_radius_m)
    |   movel([0.480649, -1.488405, -2.492708, -0.731275, 1.570796, 2.051445],accel_mss,speed_ms,0,blend_radius_m)
    |   movel([0.480991, -1.486173, -2.494642, -0.731574, 1.570796, 2.051788],accel_mss,speed_ms,0,blend_radius_m)
    |   movel([0.481470, -1.483852, -2.496643, -0.731893, 1.570796, 2.052266],accel_mss,speed_ms,0,blend_radius_m)
    |   movel([0.482087, -1.481456, -2.498701, -0.732232, 1.570796, 2.052883],accel_mss,speed_ms,0,blend_radius_m)
    |   movel([0.482851, -1.479008, -2.500794, -0.732587, 1.570796, 2.053648],accel_mss,speed_ms,0,blend_radius_m)
    |   movel([0.483763, -1.476523, -2.502909, -0.732957, 1.570796, 2.054560],accel_mss,speed_ms,0,blend_radius_m)
    |   movel([0.484830, -1.474022, -2.505028, -0.733339, 1.570796, 2.055627],accel_mss,speed_ms,0,blend_radius_m)
    |   movel([0.486057, -1.471525, -2.507134, -0.733730, 1.570796, 2.056854],accel_mss,speed_ms,0,blend_radius_m)
    |   movel([0.487449, -1.469050, -2.509211, -0.734128, 1.570796, 2.058245],accel_mss,speed_ms,0,blend_radius_m)
    |   movel([0.489008, -1.466616, -2.511245, -0.734528, 1.570796, 2.059805],accel_mss,speed_ms,0,blend_radius_m)
    |   movel([0.490739, -1.464248, -2.513215, -0.734927, 1.570796, 2.061535],accel_mss,speed_ms,0,blend_radius_m)
    |   movel([0.492647, -1.461961, -2.515109, -0.735320, 1.570796, 2.063443],accel_mss,speed_ms,0,blend_radius_m)
    |   movel([0.494736, -1.459780, -2.516907, -0.735702, 1.570796, 2.065532],accel_mss,speed_ms,0,blend_radius_m)
    |   movel([0.497007, -1.457726, -2.518594, -0.736069, 1.570796, 2.067803],accel_mss,speed_ms,0,blend_radius_m)
    |   movel([0.499467, -1.455820, -2.520154, -0.736415, 1.570796, 2.070264],accel_mss,speed_ms,0,blend_radius_m)
    |   movel([0.502114, -1.454087, -2.521567, -0.736735, 1.570796, 2.072911],accel_mss,speed_ms,0,blend_radius_m)
    |   movel([0.504952, -1.452548, -2.522818, -0.737023, 1.570796, 2.075748],accel_mss,speed_ms,0,blend_radius_m)
    |   movel([0.506085, -1.452062, -2.523213, -0.737114, 1.570796, 2.076882],accel_mss,speed_ms,0,blend_radius_m)
    |   movel([0.506646, -1.451910, -2.523336, -0.737143, 1.570796, 2.077442],accel_mss,speed_ms,0,blend_radius_m)
    |   movel([0.507180, -1.451865, -2.523372, -0.737151, 1.570796, 2.077976],accel_mss,speed_ms,0,blend_radius_m)
    |   movel([0.507850, -1.452048, -2.523224, -0.737117, 1.570796, 2.078646],accel_mss,speed_ms,0,blend_radius_m)
    |   movel([0.508305, -1.452476, -2.522877, -0.737036, 1.570796, 2.079101],accel_mss,speed_ms,0,blend_radius_m)
    |   movel([0.508559, -1.453073, -2.522392, -0.736924, 1.570796, 2.079355],accel_mss,speed_ms,0,blend_radius_m)
    |   movel([0.508624, -1.453762, -2.521832, -0.736795, 1.570796, 2.079421],accel_mss,speed_ms,0,blend_radius_m)
    |   movel([0.508371, -1.455391, -2.520505, -0.736494, 1.570796, 2.079167],accel_mss,speed_ms,0,blend_radius_m)
    |   movel([0.507807, -1.457086, -2.519119, -0.736184, 1.570796, 2.078604],accel_mss,speed_ms,0,blend_radius_m)
    |   movel([0.506383, -1.460472, -2.516337, -0.735580, 1.570796, 2.077180],accel_mss,speed_ms,0,blend_radius_m)
    |   movel([0.506259, -1.461115, -2.515807, -0.735467, 1.570796, 2.077056],accel_mss,speed_ms,0,blend_radius_m)
    |   movel([0.506393, -1.461311, -2.515645, -0.735433, 1.570796, 2.077189],accel_mss,speed_ms,0,blend_radius_m)
    |   movel([0.506705, -1.461409, -2.515565, -0.735416, 1.570796, 2.077502],accel_mss,speed_ms,0,blend_radius_m)
    |   movel([0.507835, -1.460385, -2.516409, -0.735595, 1.570796, 2.078631],accel_mss,speed_ms,0,blend_radius_m)
    |   movel([0.508922, -1.459289, -2.517311, -0.735789, 1.570796, 2.079718],accel_mss,speed_ms,0,blend_radius_m)
    |   movel([0.506690, -1.464208, -2.513247, -0.734933, 1.570796, 2.077486],accel_mss,speed_ms,0,blend_radius_m)
    |   movel([0.504647, -1.469094, -2.509174, -0.734121, 1.570796, 2.075443],accel_mss,speed_ms,0,blend_radius_m)
    |   movel([0.502794, -1.473940, -2.505097, -0.733352, 1.570796, 2.073591],accel_mss,speed_ms,0,blend_radius_m)
    |   movel([0.501130, -1.478747, -2.501017, -0.732625, 1.570796, 2.071926],accel_mss,speed_ms,0,blend_radius_m)
    |   movel([0.500482, -1.480827, -2.499240, -0.732322, 1.570796, 2.071279],accel_mss,speed_ms,0,blend_radius_m)
    |   movel([0.499986, -1.482980, -2.497394, -0.732016, 1.570796, 2.070782],accel_mss,speed_ms,0,blend_radius_m)
    |   movel([0.499855, -1.484030, -2.496490, -0.731869, 1.570796, 2.070651],accel_mss,speed_ms,0,blend_radius_m)
    |   movel([0.499835, -1.485034, -2.495625, -0.731730, 1.570796, 2.070632],accel_mss,speed_ms,0,blend_radius_m)
    |   movel([0.499953, -1.485969, -2.494818, -0.731602, 1.570796, 2.070750],accel_mss,speed_ms,0,blend_radius_m)
    |   movel([0.500234, -1.486813, -2.494088, -0.731488, 1.570796, 2.071030],accel_mss,speed_ms,0,blend_radius_m)
    |   movel([0.500540, -1.487327, -2.493643, -0.731419, 1.570796, 2.071337],accel_mss,speed_ms,0,blend_radius_m)
    |   movel([0.501409, -1.488098, -2.492975, -0.731316, 1.570796, 2.072205],accel_mss,speed_ms,0,blend_radius_m)
    |   movel([0.501954, -1.488363, -2.492745, -0.731281, 1.570796, 2.072751],accel_mss,speed_ms,0,blend_radius_m)
    |   movel([0.503221, -1.488682, -2.492468, -0.731239, 1.570796, 2.074017],accel_mss,speed_ms,0,blend_radius_m)
    |   movel([0.504669, -1.488745, -2.492413, -0.731231, 1.570796, 2.075466],accel_mss,speed_ms,0,blend_radius_m)
    |   movel([0.506229, -1.488592, -2.492546, -0.731251, 1.570796, 2.077025],accel_mss,speed_ms,0,blend_radius_m)
    |   movel([0.507834, -1.488256, -2.492838, -0.731295, 1.570796, 2.078630],accel_mss,speed_ms,0,blend_radius_m)
    |   movel([0.509415, -1.487776, -2.493254, -0.731359, 1.570796, 2.080211],accel_mss,speed_ms,0,blend_radius_m)
    |   movel([0.510902, -1.487184, -2.493767, -0.731438, 1.570796, 2.081698],accel_mss,speed_ms,0,blend_radius_m)
    |   speed_ms = 0.005
    |   movel([0.510902, -1.479192, -2.490228, -0.742968, 1.570796, 2.081698],accel_mss,speed_ms,0,blend_radius_m)
    |   speed_ms = 0.040
    |   movel([0.504315, -1.478811, -2.490555, -0.743024, 1.570796, 2.075111],accel_mss,speed_ms,0,blend_radius_m)
    |   speed_ms = 0.005
    |   movel([0.504315, -1.486806, -2.494094, -0.731489, 1.570796, 2.075111],accel_mss,speed_ms,0,blend_radius_m)
    |   speed_ms = 0.025
    |   movel([0.505537, -1.486277, -2.494552, -0.731560, 1.570796, 2.076334],accel_mss,speed_ms,0,blend_radius_m)
    |   movel([0.508048, -1.484927, -2.495717, -0.731745, 1.570796, 2.078844],accel_mss,speed_ms,0,blend_radius_m)
    |   movel([0.509310, -1.484124, -2.496410, -0.731856, 1.570796, 2.080107],accel_mss,speed_ms,0,blend_radius_m)
    |   movel([0.511786, -1.482304, -2.497974, -0.732111, 1.570796, 2.082582],accel_mss,speed_ms,0,blend_radius_m)
    |   movel([0.514121, -1.480259, -2.499726, -0.732404, 1.570796, 2.084918],accel_mss,speed_ms,0,blend_radius_m)
    |   movel([0.515205, -1.479174, -2.500652, -0.732562, 1.570796, 2.086001],accel_mss,speed_ms,0,blend_radius_m)
    |   movel([0.516215, -1.478057, -2.501605, -0.732727, 1.570796, 2.087012],accel_mss,speed_ms,0,blend_radius_m)
    |   movel([0.517967, -1.475769, -2.503549, -0.733071, 1.570796, 2.088763],accel_mss,speed_ms,0,blend_radius_m)
    |   movel([0.518685, -1.474614, -2.504528, -0.733248, 1.570796, 2.089481],accel_mss,speed_ms,0,blend_radius_m)
    |   movel([0.519277, -1.473465, -2.505498, -0.733425, 1.570796, 2.090073],accel_mss,speed_ms,0,blend_radius_m)
    |   movel([0.519733, -1.472331, -2.506455, -0.733603, 1.570796, 2.090530],accel_mss,speed_ms,0,blend_radius_m)
    |   movel([0.520040, -1.471221, -2.507390, -0.733779, 1.570796, 2.090837],accel_mss,speed_ms,0,blend_radius_m)
    |   movel([0.520253, -1.469872, -2.508522, -0.733995, 1.570796, 2.091049],accel_mss,speed_ms,0,blend_radius_m)
    |   movel([0.520313, -1.468570, -2.509613, -0.734206, 1.570796, 2.091109],accel_mss,speed_ms,0,blend_radius_m)
    |   movel([0.520194, -1.467346, -2.510636, -0.734407, 1.570796, 2.090990],accel_mss,speed_ms,0,blend_radius_m)
    |   movel([0.519870, -1.466239, -2.511559, -0.734591, 1.570796, 2.090666],accel_mss,speed_ms,0,blend_radius_m)
    |   movel([0.519315, -1.465282, -2.512355, -0.734751, 1.570796, 2.090111],accel_mss,speed_ms,0,blend_radius_m)
    |   movel([0.518505, -1.464514, -2.512994, -0.734881, 1.570796, 2.089301],accel_mss,speed_ms,0,blend_radius_m)
    |   movel([0.517413, -1.463971, -2.513444, -0.734974, 1.570796, 2.088209],accel_mss,speed_ms,0,blend_radius_m)
    |   movel([0.516017, -1.463685, -2.513681, -0.735023, 1.570796, 2.086813],accel_mss,speed_ms,0,blend_radius_m)
    |   movel([0.514950, -1.463686, -2.513680, -0.735022, 1.570796, 2.085747],accel_mss,speed_ms,0,blend_radius_m)
    |   movel([0.513820, -1.463866, -2.513531, -0.734992, 1.570796, 2.084616],accel_mss,speed_ms,0,blend_radius_m)
    |   movel([0.512668, -1.464211, -2.513245, -0.734933, 1.570796, 2.083464],accel_mss,speed_ms,0,blend_radius_m)
    |   movel([0.511531, -1.464705, -2.512835, -0.734849, 1.570796, 2.082327],accel_mss,speed_ms,0,blend_radius_m)
    |   movel([0.510447, -1.465335, -2.512311, -0.734743, 1.570796, 2.081243],accel_mss,speed_ms,0,blend_radius_m)
    |   movel([0.509455, -1.466086, -2.511687, -0.734617, 1.570796, 2.080251],accel_mss,speed_ms,0,blend_radius_m)
    |   movel([0.508594, -1.466942, -2.510973, -0.734474, 1.570796, 2.079391],accel_mss,speed_ms,0,blend_radius_m)
    |   movel([0.507900, -1.467889, -2.510182, -0.734318, 1.570796, 2.078696],accel_mss,speed_ms,0,blend_radius_m)
    |   speed_ms = 0.005
    |   movel([0.507900, -1.459742, -2.506566, -0.746082, 1.570796, 2.078696],accel_mss,speed_ms,0,blend_radius_m)
    |   speed_ms = 0.040
    |   # Splitting Linear movement in 2 (instruction 399: MoveL 378)
    |   movel([0.523348, -1.483026, -2.486939, -0.742424, 1.570796, 2.094144],accel_mss,speed_ms,0,blend_radius_m)
    |   movel([0.537863, -1.506106, -2.466651, -0.739632, 1.570796, 2.108659],accel_mss,speed_ms,0,blend_radius_m)
    |   speed_ms = 0.005
    |   movel([0.537863, -1.513881, -2.470084, -0.728424, 1.570796, 2.108659],accel_mss,speed_ms,0,blend_radius_m)
    |   speed_ms = 0.025
    |   movel([0.534804, -1.518746, -2.465646, -0.727997, 1.570796, 2.105600],accel_mss,speed_ms,0,blend_radius_m)
    |   movel([0.533121, -1.521109, -2.463476, -0.727804, 1.570796, 2.103918],accel_mss,speed_ms,0,blend_radius_m)
    |   movel([0.532179, -1.522267, -2.462410, -0.727712, 1.570796, 2.102975],accel_mss,speed_ms,0,blend_radius_m)
    |   movel([0.531146, -1.523403, -2.461362, -0.727624, 1.570796, 2.101942],accel_mss,speed_ms,0,blend_radius_m)
    |   movel([0.529945, -1.524547, -2.460304, -0.727538, 1.570796, 2.100741],accel_mss,speed_ms,0,blend_radius_m)
    |   movel([0.529289, -1.525058, -2.459830, -0.727500, 1.570796, 2.100085],accel_mss,speed_ms,0,blend_radius_m)
    |   movel([0.528582, -1.525499, -2.459422, -0.727468, 1.570796, 2.099378],accel_mss,speed_ms,0,blend_radius_m)
    |   movel([0.529133, -1.524304, -2.460528, -0.727556, 1.570796, 2.099929],accel_mss,speed_ms,0,blend_radius_m)
    |   movel([0.529482, -1.523112, -2.461630, -0.727647, 1.570796, 2.100279],accel_mss,speed_ms,0,blend_radius_m)
    |   movel([0.529474, -1.522730, -2.461983, -0.727676, 1.570796, 2.100270],accel_mss,speed_ms,0,blend_radius_m)
    |   movel([0.529326, -1.522627, -2.462078, -0.727684, 1.570796, 2.100123],accel_mss,speed_ms,0,blend_radius_m)
    |   movel([0.529110, -1.522609, -2.462095, -0.727685, 1.570796, 2.099906],accel_mss,speed_ms,0,blend_radius_m)
    |   movel([0.528595, -1.522751, -2.461963, -0.727674, 1.570796, 2.099391],accel_mss,speed_ms,0,blend_radius_m)
    |   movel([0.527773, -1.523173, -2.461574, -0.727642, 1.570796, 2.098570],accel_mss,speed_ms,0,blend_radius_m)
    |   movel([0.527042, -1.523682, -2.461104, -0.727603, 1.570796, 2.097839],accel_mss,speed_ms,0,blend_radius_m)
    |   movel([0.526387, -1.524259, -2.460570, -0.727560, 1.570796, 2.097183],accel_mss,speed_ms,0,blend_radius_m)
    |   movel([0.525792, -1.524887, -2.459990, -0.727513, 1.570796, 2.096588],accel_mss,speed_ms,0,blend_radius_m)
    |   movel([0.523657, -1.527569, -2.457500, -0.727320, 1.570796, 2.094453],accel_mss,speed_ms,0,blend_radius_m)
    |   movel([0.522328, -1.529102, -2.456072, -0.727215, 1.570796, 2.093124],accel_mss,speed_ms,0,blend_radius_m)
    |   movel([0.520904, -1.530578, -2.454693, -0.727118, 1.570796, 2.091700],accel_mss,speed_ms,0,blend_radius_m)
    |   movel([0.519366, -1.531969, -2.453391, -0.727029, 1.570796, 2.090162],accel_mss,speed_ms,0,blend_radius_m)
    |   movel([0.517701, -1.533238, -2.452200, -0.726951, 1.570796, 2.088497],accel_mss,speed_ms,0,blend_radius_m)
    |   movel([0.518592, -1.531972, -2.453389, -0.727029, 1.570796, 2.089388],accel_mss,speed_ms,0,blend_radius_m)
    |   movel([0.519175, -1.530653, -2.454623, -0.727113, 1.570796, 2.089972],accel_mss,speed_ms,0,blend_radius_m)
    |   movel([0.519249, -1.530320, -2.454934, -0.727134, 1.570796, 2.090045],accel_mss,speed_ms,0,blend_radius_m)
    |   movel([0.519182, -1.530039, -2.455197, -0.727153, 1.570796, 2.089978],accel_mss,speed_ms,0,blend_radius_m)
    |   movel([0.518981, -1.529919, -2.455309, -0.727161, 1.570796, 2.089777],accel_mss,speed_ms,0,blend_radius_m)
    |   movel([0.518695, -1.529909, -2.455318, -0.727161, 1.570796, 2.089492],accel_mss,speed_ms,0,blend_radius_m)
    |   movel([0.518041, -1.530107, -2.455134, -0.727148, 1.570796, 2.088838],accel_mss,speed_ms,0,blend_radius_m)
    |   movel([0.517247, -1.530525, -2.454743, -0.727121, 1.570796, 2.088044],accel_mss,speed_ms,0,blend_radius_m)
    |   movel([0.516500, -1.531034, -2.454266, -0.727088, 1.570796, 2.087296],accel_mss,speed_ms,0,blend_radius_m)
    |   movel([0.515121, -1.532230, -2.453147, -0.727013, 1.570796, 2.085917],accel_mss,speed_ms,0,blend_radius_m)
    |   movel([0.512588, -1.534774, -2.450755, -0.726860, 1.570796, 2.083384],accel_mss,speed_ms,0,blend_radius_m)
    |   movel([0.511075, -1.536112, -2.449494, -0.726783, 1.570796, 2.081871],accel_mss,speed_ms,0,blend_radius_m)
    |   movel([0.509482, -1.537370, -2.448304, -0.726714, 1.570796, 2.080278],accel_mss,speed_ms,0,blend_radius_m)
    |   movel([0.507801, -1.538507, -2.447228, -0.726654, 1.570796, 2.078597],accel_mss,speed_ms,0,blend_radius_m)
    |   movel([0.506025, -1.539481, -2.446304, -0.726604, 1.570796, 2.076821],accel_mss,speed_ms,0,blend_radius_m)
    |   movel([0.506593, -1.538824, -2.446928, -0.726638, 1.570796, 2.077389],accel_mss,speed_ms,0,blend_radius_m)
    |   movel([0.507483, -1.537432, -2.448246, -0.726711, 1.570796, 2.078279],accel_mss,speed_ms,0,blend_radius_m)
    |   movel([0.507792, -1.536717, -2.448922, -0.726750, 1.570796, 2.078589],accel_mss,speed_ms,0,blend_radius_m)
    |   movel([0.507859, -1.536388, -2.449233, -0.726768, 1.570796, 2.078655],accel_mss,speed_ms,0,blend_radius_m)
    |   movel([0.507713, -1.536176, -2.449433, -0.726780, 1.570796, 2.078509],accel_mss,speed_ms,0,blend_radius_m)
    |   movel([0.507336, -1.536230, -2.449382, -0.726777, 1.570796, 2.078132],accel_mss,speed_ms,0,blend_radius_m)
    |   movel([0.506369, -1.536616, -2.449017, -0.726755, 1.570796, 2.077165],accel_mss,speed_ms,0,blend_radius_m)
    |   movel([0.505468, -1.537086, -2.448573, -0.726730, 1.570796, 2.076264],accel_mss,speed_ms,0,blend_radius_m)
    |   movel([0.503783, -1.538190, -2.447528, -0.726671, 1.570796, 2.074579],accel_mss,speed_ms,0,blend_radius_m)
    |   movel([0.502119, -1.539347, -2.446431, -0.726611, 1.570796, 2.072916],accel_mss,speed_ms,0,blend_radius_m)
    |   movel([0.501243, -1.539886, -2.445919, -0.726584, 1.570796, 2.072040],accel_mss,speed_ms,0,blend_radius_m)
    |   movel([0.500309, -1.540369, -2.445461, -0.726560, 1.570796, 2.071105],accel_mss,speed_ms,0,blend_radius_m)
    |   movel([0.497992, -1.541360, -2.444518, -0.726512, 1.570796, 2.068789],accel_mss,speed_ms,0,blend_radius_m)
    |   movel([0.495656, -1.542234, -2.443684, -0.726471, 1.570796, 2.066453],accel_mss,speed_ms,0,blend_radius_m)
    |   movel([0.493314, -1.543007, -2.442947, -0.726436, 1.570796, 2.064111],accel_mss,speed_ms,0,blend_radius_m)
    |   movel([0.490972, -1.543698, -2.442286, -0.726405, 1.570796, 2.061768],accel_mss,speed_ms,0,blend_radius_m)
    |   speed_ms = 0.005
    |   movel([0.490972, -1.536166, -2.438968, -0.737255, 1.570796, 2.061768],accel_mss,speed_ms,0,blend_radius_m)
    |   speed_ms = 0.040
    |   movel([0.487780, -1.510169, -2.462992, -0.739227, 1.570796, 2.058576],accel_mss,speed_ms,0,blend_radius_m)
    |   speed_ms = 0.005
    |   movel([0.487780, -1.517912, -2.466409, -0.728068, 1.570796, 2.058576],accel_mss,speed_ms,0,blend_radius_m)
    |   speed_ms = 0.025
    |   movel([0.488572, -1.517575, -2.466717, -0.728097, 1.570796, 2.059368],accel_mss,speed_ms,0,blend_radius_m)
    |   movel([0.489350, -1.517128, -2.467126, -0.728135, 1.570796, 2.060146],accel_mss,speed_ms,0,blend_radius_m)
    |   movel([0.490888, -1.516039, -2.468120, -0.728230, 1.570796, 2.061684],accel_mss,speed_ms,0,blend_radius_m)
    |   movel([0.492434, -1.514904, -2.469154, -0.728331, 1.570796, 2.063230],accel_mss,speed_ms,0,blend_radius_m)
    |   movel([0.493224, -1.514400, -2.469612, -0.728377, 1.570796, 2.064021],accel_mss,speed_ms,0,blend_radius_m)
    |   movel([0.494032, -1.513985, -2.469990, -0.728415, 1.570796, 2.064828],accel_mss,speed_ms,0,blend_radius_m)
    |   movel([0.494623, -1.513764, -2.470190, -0.728435, 1.570796, 2.065419],accel_mss,speed_ms,0,blend_radius_m)
    |   movel([0.495063, -1.513684, -2.470262, -0.728442, 1.570796, 2.065860],accel_mss,speed_ms,0,blend_radius_m)
    |   movel([0.495369, -1.513727, -2.470223, -0.728438, 1.570796, 2.066165],accel_mss,speed_ms,0,blend_radius_m)
    |   movel([0.495556, -1.513878, -2.470087, -0.728425, 1.570796, 2.066352],accel_mss,speed_ms,0,blend_radius_m)
    |   movel([0.495622, -1.514444, -2.469572, -0.728373, 1.570796, 2.066419],accel_mss,speed_ms,0,blend_radius_m)
    |   movel([0.495380, -1.515256, -2.468833, -0.728300, 1.570796, 2.066176],accel_mss,speed_ms,0,blend_radius_m)
    |   movel([0.494420, -1.517121, -2.467132, -0.728136, 1.570796, 2.065216],accel_mss,speed_ms,0,blend_radius_m)
    |   movel([0.493590, -1.518486, -2.465884, -0.728019, 1.570796, 2.064386],accel_mss,speed_ms,0,blend_radius_m)
    |   movel([0.495203, -1.517431, -2.466849, -0.728109, 1.570796, 2.065999],accel_mss,speed_ms,0,blend_radius_m)
    |   movel([0.496592, -1.516279, -2.467900, -0.728209, 1.570796, 2.067388],accel_mss,speed_ms,0,blend_radius_m)
    |   movel([0.497820, -1.515050, -2.469020, -0.728318, 1.570796, 2.068616],accel_mss,speed_ms,0,blend_radius_m)
    |   movel([0.498939, -1.513767, -2.470188, -0.728435, 1.570796, 2.069735],accel_mss,speed_ms,0,blend_radius_m)
    |   movel([0.502214, -1.509791, -2.473786, -0.728812, 1.570796, 2.073011],accel_mss,speed_ms,0,blend_radius_m)
    |   movel([0.503467, -1.508496, -2.474952, -0.728941, 1.570796, 2.074264],accel_mss,speed_ms,0,blend_radius_m)
    |   movel([0.504042, -1.508033, -2.475369, -0.728987, 1.570796, 2.074839],accel_mss,speed_ms,0,blend_radius_m)
    |   movel([0.504505, -1.507825, -2.475555, -0.729008, 1.570796, 2.075301],accel_mss,speed_ms,0,blend_radius_m)
    |   movel([0.504864, -1.507828, -2.475553, -0.729008, 1.570796, 2.075660],accel_mss,speed_ms,0,blend_radius_m)
    |   movel([0.505123, -1.508000, -2.475398, -0.728991, 1.570796, 2.075919],accel_mss,speed_ms,0,blend_radius_m)
    |   movel([0.505294, -1.508296, -2.475132, -0.728961, 1.570796, 2.076091],accel_mss,speed_ms,0,blend_radius_m)
    |   movel([0.505381, -1.508672, -2.474794, -0.728923, 1.570796, 2.076177],accel_mss,speed_ms,0,blend_radius_m)
    |   movel([0.505338, -1.509493, -2.474054, -0.728842, 1.570796, 2.076134],accel_mss,speed_ms,0,blend_radius_m)
    |   movel([0.505014, -1.510325, -2.473304, -0.728760, 1.570796, 2.075810],accel_mss,speed_ms,0,blend_radius_m)
    |   movel([0.504439, -1.511358, -2.472370, -0.728660, 1.570796, 2.075235],accel_mss,speed_ms,0,blend_radius_m)
    |   movel([0.503263, -1.513232, -2.470673, -0.728484, 1.570796, 2.074059],accel_mss,speed_ms,0,blend_radius_m)
    |   movel([0.505626, -1.510620, -2.473038, -0.728732, 1.570796, 2.076422],accel_mss,speed_ms,0,blend_radius_m)
    |   movel([0.506698, -1.509260, -2.474264, -0.728865, 1.570796, 2.077494],accel_mss,speed_ms,0,blend_radius_m)
    |   movel([0.508605, -1.506453, -2.476787, -0.729149, 1.570796, 2.079402],accel_mss,speed_ms,0,blend_radius_m)
    |   movel([0.509431, -1.505018, -2.478072, -0.729299, 1.570796, 2.080227],accel_mss,speed_ms,0,blend_radius_m)
    |   movel([0.510811, -1.502110, -2.480666, -0.729613, 1.570796, 2.081607],accel_mss,speed_ms,0,blend_radius_m)
    |   speed_ms = 0.005
    |   movel([0.510811, -1.494239, -2.477187, -0.740963, 1.570796, 2.081607],accel_mss,speed_ms,0,blend_radius_m)
    |   speed_ms = 0.040
    |   movel([0.497117, -1.501666, -2.470618, -0.740104, 1.570796, 2.067913],accel_mss,speed_ms,0,blend_radius_m)
    |   speed_ms = 0.005
    |   movel([0.497117, -1.509478, -2.474068, -0.728843, 1.570796, 2.067913],accel_mss,speed_ms,0,blend_radius_m)
    |   speed_ms = 0.025
    |   movel([0.495257, -1.510649, -2.473012, -0.728729, 1.570796, 2.066053],accel_mss,speed_ms,0,blend_radius_m)
    |   movel([0.493461, -1.511915, -2.471867, -0.728607, 1.570796, 2.064257],accel_mss,speed_ms,0,blend_radius_m)
    |   movel([0.489912, -1.514496, -2.469525, -0.728368, 1.570796, 2.060708],accel_mss,speed_ms,0,blend_radius_m)
    |   movel([0.488066, -1.515701, -2.468428, -0.728260, 1.570796, 2.058863],accel_mss,speed_ms,0,blend_radius_m)
    |   movel([0.486153, -1.516758, -2.467464, -0.728167, 1.570796, 2.056949],accel_mss,speed_ms,0,blend_radius_m)
    |   movel([0.484199, -1.517579, -2.466714, -0.728096, 1.570796, 2.054996],accel_mss,speed_ms,0,blend_radius_m)
    |   movel([0.483218, -1.517873, -2.466445, -0.728071, 1.570796, 2.054014],accel_mss,speed_ms,0,blend_radius_m)
    |   movel([0.482238, -1.518076, -2.466259, -0.728054, 1.570796, 2.053034],accel_mss,speed_ms,0,blend_radius_m)
    |   movel([0.483018, -1.517797, -2.466514, -0.728078, 1.570796, 2.053815],accel_mss,speed_ms,0,blend_radius_m)
    |   movel([0.483969, -1.517228, -2.467035, -0.728127, 1.570796, 2.054765],accel_mss,speed_ms,0,blend_radius_m)
    |   movel([0.484967, -1.516459, -2.467736, -0.728193, 1.570796, 2.055763],accel_mss,speed_ms,0,blend_radius_m)
    |   movel([0.485881, -1.515585, -2.468533, -0.728270, 1.570796, 2.056677],accel_mss,speed_ms,0,blend_radius_m)
    |   movel([0.486585, -1.514696, -2.469343, -0.728350, 1.570796, 2.057381],accel_mss,speed_ms,0,blend_radius_m)
    |   movel([0.486814, -1.514276, -2.469725, -0.728388, 1.570796, 2.057611],accel_mss,speed_ms,0,blend_radius_m)
    |   movel([0.486945, -1.513888, -2.470078, -0.728424, 1.570796, 2.057741],accel_mss,speed_ms,0,blend_radius_m)
    |   movel([0.486958, -1.513541, -2.470392, -0.728455, 1.570796, 2.057755],accel_mss,speed_ms,0,blend_radius_m)
    |   movel([0.486836, -1.513251, -2.470656, -0.728482, 1.570796, 2.057632],accel_mss,speed_ms,0,blend_radius_m)
    |   movel([0.486566, -1.513027, -2.470859, -0.728503, 1.570796, 2.057362],accel_mss,speed_ms,0,blend_radius_m)
    |   movel([0.486127, -1.512881, -2.470991, -0.728517, 1.570796, 2.056923],accel_mss,speed_ms,0,blend_radius_m)
    |   movel([0.485294, -1.512904, -2.470970, -0.728514, 1.570796, 2.056090],accel_mss,speed_ms,0,blend_radius_m)
    |   movel([0.481486, -1.513751, -2.470201, -0.728436, 1.570796, 2.052282],accel_mss,speed_ms,0,blend_radius_m)
    |   movel([0.479925, -1.513965, -2.470008, -0.728417, 1.570796, 2.050722],accel_mss,speed_ms,0,blend_radius_m)
    |   movel([0.478382, -1.514060, -2.469921, -0.728408, 1.570796, 2.049179],accel_mss,speed_ms,0,blend_radius_m)
    |   movel([0.476919, -1.514007, -2.469969, -0.728413, 1.570796, 2.047715],accel_mss,speed_ms,0,blend_radius_m)
    |   movel([0.475600, -1.513769, -2.470186, -0.728435, 1.570796, 2.046397],accel_mss,speed_ms,0,blend_radius_m)
    |   movel([0.474488, -1.513312, -2.470600, -0.728477, 1.570796, 2.045285],accel_mss,speed_ms,0,blend_radius_m)
    |   movel([0.473651, -1.512599, -2.471247, -0.728543, 1.570796, 2.044447],accel_mss,speed_ms,0,blend_radius_m)
    |   movel([0.473950, -1.512766, -2.471095, -0.728527, 1.570796, 2.044746],accel_mss,speed_ms,0,blend_radius_m)
    |   movel([0.474432, -1.512811, -2.471055, -0.728523, 1.570796, 2.045228],accel_mss,speed_ms,0,blend_radius_m)
    |   movel([0.475729, -1.512633, -2.471216, -0.728540, 1.570796, 2.046525],accel_mss,speed_ms,0,blend_radius_m)
    |   movel([0.477102, -1.512257, -2.471557, -0.728575, 1.570796, 2.047899],accel_mss,speed_ms,0,blend_radius_m)
    |   movel([0.478108, -1.511875, -2.471903, -0.728611, 1.570796, 2.048905],accel_mss,speed_ms,0,blend_radius_m)
    |   movel([0.478780, -1.511488, -2.472253, -0.728648, 1.570796, 2.049577],accel_mss,speed_ms,0,blend_radius_m)
    |   movel([0.479133, -1.511140, -2.472568, -0.728681, 1.570796, 2.049929],accel_mss,speed_ms,0,blend_radius_m)
